RoboDK station: kr30 cnc 070119 curve 7 axis test.rdk

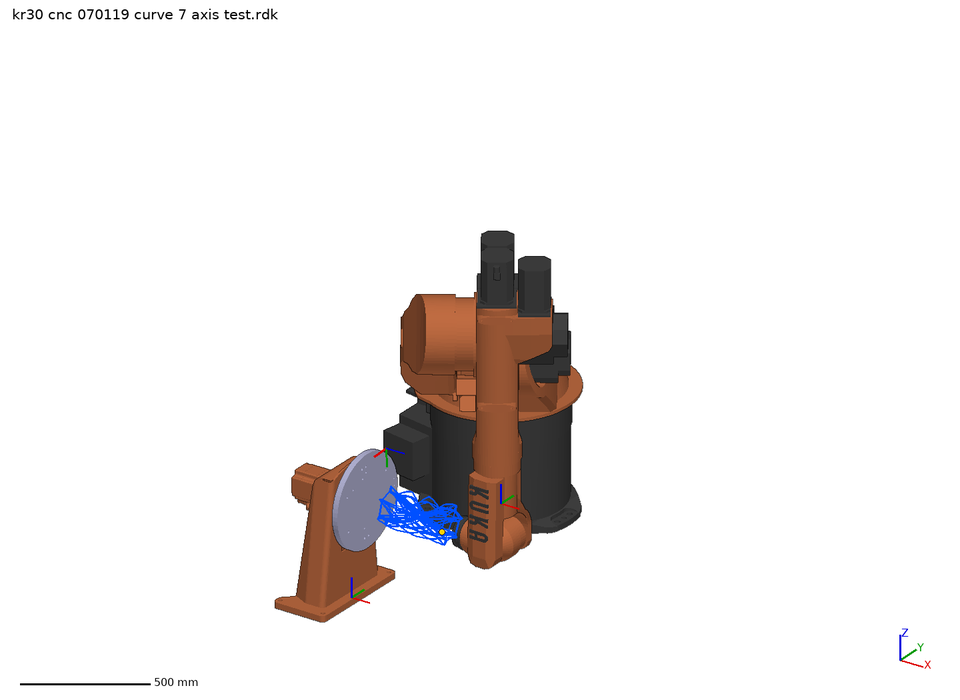
[picture v0: the station drawn from its stored meshes, robots at their saved joint values, targets as dots, program paths as lines]
Station kr30 cnc 070119 curve 7 axis test. Poses are relative to the parent item; angles as X-Y-Z fixed-axis rotations.
  - machining project Curve settings: C:/Temp/temp3/RhinoProject.stl | rotZ(0) | rotX(0)*rotY(0) | rotz(0) | onStart | onPathStart | onApproach | onPoint | onRetract | onFinish | onPathFinish
  - frame KUKA KP1 MD250 Base at (0, 1000, 0) mm
    - robot KUKA KP1 MD250: 1 axes, payload 250 kg
        modified DH rows (alpha deg, a mm, theta deg, d mm): 0, 0, 0, 0
        base shift (73.5, 0, 432) mm, rotated rx 0 ry 90 rz 0 deg
        joint limits [-3600] to [3600]; home [0]; saved at [-1886.749]
      - frame Reference Rhino at (0, -260, 100) mm
        - object RhinoPart at (0, 0, 0) mm
  - frame KUKA KR 30 HA Base at (0, 2000, 0) mm
    - robot KUKA KR 30 HA: 6 axes, payload 30 kg, reach 2033 mm, repeatability 0.05 mm, weight 665 kg
        modified DH rows (alpha deg, a mm, theta deg, d mm): 0, 0, 0, 815; -90, 350, 0, 0; 0, 850, -90, 0; -90, 145, 0, 820; 90, 0, 0, 0; -90, 0, 180, 170
        joint limits [-185, -135, -120, -350, -119, -350] to [185, 35, 158, 350, 119, 350]; home [0, -90, 90, 0, 0, 0]; saved at [55.744, -30.783, 121.676, 55.747, 89.498, 89.262]
      - tool Tool 1, TCP at (0, 0, 200) mm
  - machining project RhinoPart Settings: rotZ(0) | rotX(0)*rotY(0) | rotz(0) | onStart | onPathStart | onApproach | onPoint | onRetract | onFinish | onPathFinish
  - program RhinoPart (1340 instructions, listed below)
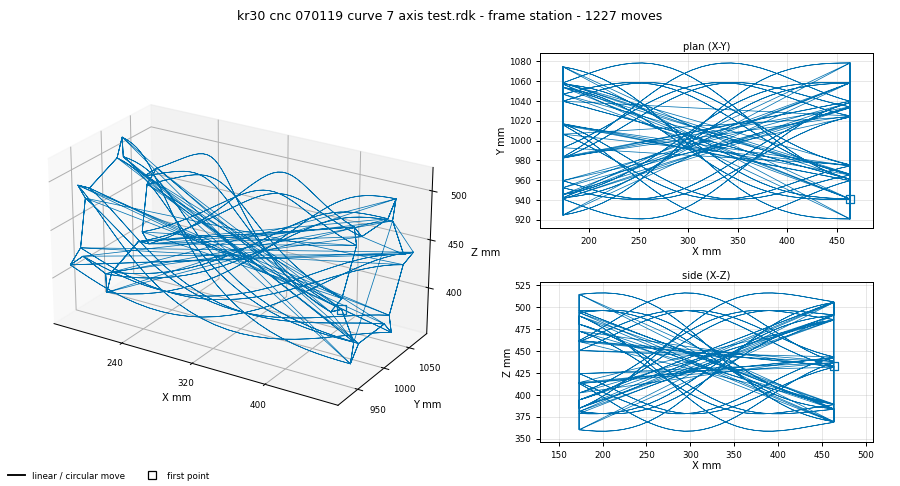
[picture p0: tool path of kr30 cnc 070119 curve 7 axis test.rdk in frame station, 1227 of 1227 moves have a stored position in this frame; points joined in program order, loops and branches not executed]

--- program RhinoPart (robot KUKA KR 30 HA) ---
  Set Ref.: Reference Rhino
  Set Tool: Tool 1
  Show Tool 1
  Set speed (1000.0 mm/s)
  MoveJ 1 to (58.93, 255.88, 290) mm, rotated rx -180 ry 0 rz -94 deg; joints [50.189, -25.769, 112.866, 50.225, 91.858, 92.231, 4.002]
  MoveL 2 to (58.93, 255.88, 290) mm, rotated rx -180 ry 0 rz -94 deg; joints [50.189, -25.769, 112.866, 50.225, 91.858, 92.231, 4.002]
  MoveL 3 to (58.93, 255.88, 290) mm, rotated rx -180 ry 0 rz -94 deg; joints [50.189, -25.769, 112.866, 50.225, 91.858, 92.231, 4.002]
  Set speed (60.0 mm/s)
  MoveL 4 to (37.11, 300.24, 290) mm, rotated rx 180 ry 0 rz -42.69 deg; joints [50.189, -26.061, 113.024, 50.228, 91.944, 92.334, -47.315]
  MoveL 5 to (-37.11, 208.63, 290) mm, rotated rx -180 ry 0 rz 144.16 deg; joints [50.189, -25.479, 112.707, 50.222, 91.774, 92.13, 125.844]
  Set speed (60.0 mm/s)
  MoveL 6 to (-58.93, 252.99, 290) mm, rotated rx -180 ry 0 rz 96.78 deg; joints [50.189, -25.75, 112.856, 50.225, 91.853, 92.224, 173.216]
  MoveL 7 to (21.11, 199.39, 290) mm, rotated rx -180 ry 0 rz -160.79 deg; joints [50.189, -25.425, 112.677, 50.221, 91.759, 92.111, 70.794]
  Set speed (60.0 mm/s)
  MoveL 8 to (34.79, 183.72, 290) mm, rotated rx -180 ry 0 rz -155.49 deg; joints [50.189, -24.101, 111.933, 50.209, 91.388, 91.665, 65.485]
  MoveL 9 to (21.11, 199.39, 290) mm, rotated rx -180 ry 0 rz -160.79 deg; joints [50.189, -25.425, 112.677, 50.221, 91.759, 92.111, 70.794]
  Set speed (60.0 mm/s)
  MoveL 10 to (-28.22, 202.67, 290) mm, rotated rx -180 ry 0 rz 153.79 deg; joints [50.189, -25.444, 112.688, 50.221, 91.764, 92.118, 116.207]
  MoveL 11 to (-43.85, 188.95, 290) mm, rotated rx -180 ry 0 rz 148.32 deg; joints [50.189, -24.124, 111.947, 50.209, 91.394, 91.673, 121.679]
  Set speed (60.0 mm/s)
  MoveL 12 to (-28.22, 202.67, 290) mm, rotated rx -180 ry 0 rz 153.79 deg; joints [50.189, -25.444, 112.688, 50.221, 91.764, 92.118, 116.207]
  MoveL 13 to (-43.85, 188.95, 290) mm, rotated rx -180 ry 0 rz 148.32 deg; joints [50.189, -24.124, 111.947, 50.209, 91.394, 91.673, 121.679]
  Set speed (60.0 mm/s)
  MoveL 14 to (-37.11, 208.63, 290) mm, rotated rx -180 ry 0 rz 144.16 deg; joints [50.189, -25.479, 112.707, 50.222, 91.774, 92.13, 125.844]
  MoveL 15 to (-78.63, 259.66, 290) mm, rotated rx -180 ry 0 rz 90.25 deg; joints [50.189, -24.451, 112.133, 50.212, 91.484, 91.781, 179.755]
  Set speed (60.0 mm/s)
  MoveL 16 to (-58.93, 252.99, 290) mm, rotated rx -180 ry 0 rz 96.78 deg; joints [50.189, -25.75, 112.856, 50.225, 91.853, 92.224, 173.216]
  MoveL 17 to (-78.63, 259.66, 290) mm, rotated rx -180 ry 0 rz 90.25 deg; joints [50.189, -24.451, 112.133, 50.212, 91.484, 91.781, 179.755]
  Set speed (60.0 mm/s)
  MoveL 18 to (-58.22, 263.67, 290) mm, rotated rx -180 ry 0 rz 86.39 deg; joints [50.189, -25.818, 112.893, 50.226, 91.873, 92.248, 183.606]
  MoveL 19 to (-30.72, 304.75, 290) mm, rotated rx -180 ry 0 rz 34.47 deg; joints [50.189, -26.092, 113.041, 50.229, 91.953, 92.345, 235.533]
  Set speed (60.0 mm/s)
  MoveL 20 to (-58.22, 263.67, 290) mm, rotated rx -180 ry 0 rz 86.39 deg; joints [50.189, -25.818, 112.893, 50.226, 91.873, 92.248, 183.606]
  MoveL 21 to (-30.72, 304.75, 290) mm, rotated rx -180 ry 0 rz 34.47 deg; joints [50.189, -26.092, 113.041, 50.229, 91.953, 92.345, 235.533]
  Set speed (60.0 mm/s)
  MoveL 22 to (-34.79, 325.15, 290) mm, rotated rx -180 ry 0 rz 28.1 deg; joints [50.189, -24.773, 112.315, 50.215, 91.574, 91.889, 241.899]
  MoveL 23 to (-21.11, 309.47, 290) mm, rotated rx 180 ry 0 rz 23.11 deg; joints [50.189, -26.125, 113.059, 50.229, 91.963, 92.356, 246.89]
  Set speed (60.0 mm/s)
  MoveL 24 to (-34.79, 325.15, 290) mm, rotated rx -180 ry 0 rz 28.1 deg; joints [50.189, -24.773, 112.315, 50.215, 91.574, 91.889, 241.899]
  MoveL 25 to (-21.11, 309.47, 290) mm, rotated rx 180 ry 0 rz 23.11 deg; joints [50.189, -26.125, 113.059, 50.229, 91.963, 92.356, 246.89]
  Set speed (60.0 mm/s)
  MoveL 26 to (28.22, 306.19, 290) mm, rotated rx -180 ry 0 rz -31.42 deg; joints [50.189, -26.102, 113.046, 50.229, 91.956, 92.348, 301.418]
  MoveL 27 to (43.85, 319.91, 290) mm, rotated rx -180 ry 0 rz -36.2 deg; joints [50.189, -24.747, 112.3, 50.214, 91.566, 91.88, 306.197]
  Set speed (60.0 mm/s)
  MoveL 28 to (28.22, 306.19, 290) mm, rotated rx -180 ry 0 rz -31.42 deg; joints [50.189, -26.102, 113.046, 50.229, 91.956, 92.348, 301.418]
  MoveL 29 to (43.85, 319.91, 290) mm, rotated rx -180 ry 0 rz -36.2 deg; joints [50.189, -24.747, 112.3, 50.214, 91.566, 91.88, 306.197]
  Set speed (60.0 mm/s)
  MoveL 30 to (37.11, 300.24, 290) mm, rotated rx 180 ry 0 rz -42.69 deg; joints [50.189, -26.061, 113.024, 50.228, 91.944, 92.334, 312.685]
  MoveL 31 to (78.63, 249.2, 290) mm, rotated rx -180 ry 0 rz -97.82 deg; joints [50.189, -24.402, 112.105, 50.211, 91.47, 91.765, 367.819]
  Set speed (60.0 mm/s)
  MoveL 32 to (58.93, 255.88, 290) mm, rotated rx 180 ry 0 rz -94 deg; joints [50.189, -25.769, 112.866, 50.225, 91.858, 92.231, 364.002]
  MoveL 33 to (78.63, 249.2, 290) mm, rotated rx -180 ry 0 rz -97.82 deg; joints [50.189, -24.402, 112.105, 50.211, 91.47, 91.765, 367.819]
  Set speed (60.0 mm/s)
  MoveL 34 to (58.22, 245.2, 290) mm, rotated rx 180 ry 0 rz -104.27 deg; joints [50.189, -25.701, 112.829, 50.224, 91.839, 92.207, 374.265]
  MoveL 35 to (30.72, 204.12, 290) mm, rotated rx 180 ry 0 rz -151.2 deg; joints [50.189, -25.453, 112.693, 50.221, 91.767, 92.121, 421.204]
  Set speed (60.0 mm/s)
  MoveL 36 to (58.22, 245.2, 290) mm, rotated rx 180 ry 0 rz -104.27 deg; joints [50.189, -25.701, 112.829, 50.224, 91.839, 92.207, 374.265]
  MoveL 37 to (30.72, 204.12, 290) mm, rotated rx 180 ry 0 rz -151.2 deg; joints [50.189, -25.453, 112.693, 50.221, 91.767, 92.121, 421.204]
  Set speed (60.0 mm/s)
  MoveL 38 to (34.79, 183.72, 290) mm, rotated rx -180 ry 0 rz -155.49 deg; joints [50.189, -24.101, 111.933, 50.209, 91.388, 91.665, 425.485]
  MoveL 39 to (-37.62, 299.82, 0) mm, rotated rx -180 ry 0 rz 43.38 deg; joints [61.476, -27.63, 125.243, 61.688, 86.373, 83.302, 586.623]
  Set speed (60.0 mm/s)
  MoveL 40 to (10.16, 312.5, 0) mm, rotated rx -180 ry 0 rz -10.95 deg; joints [61.476, -27.728, 125.294, 61.686, 86.395, 83.343, 640.953]
  MoveL 41 to (-37.62, 299.82, 0) mm, rotated rx 180 ry 0 rz 43.38 deg; joints [61.476, -27.63, 125.243, 61.688, 86.373, 83.302, 586.623]
  Set speed (60.0 mm/s)
  MoveL 42 to (-55.59, 310.29, 0) mm, rotated rx 180 ry 0 rz 47.87 deg; joints [61.476, -26.133, 124.437, 61.729, 86.045, 82.692, 582.13]
  MoveL 43 to (-45.21, 292.27, 0) mm, rotated rx -180 ry 0 rz 54.48 deg; joints [61.476, -27.574, 125.213, 61.69, 86.36, 83.279, 575.516]
  Set speed (60.0 mm/s)
  MoveL 44 to (-55.59, 310.29, 0) mm, rotated rx 180 ry 0 rz 47.87 deg; joints [61.476, -26.133, 124.437, 61.729, 86.045, 82.692, 582.13]
  MoveL 45 to (-45.21, 292.27, 0) mm, rotated rx -180 ry 0 rz 54.48 deg; joints [61.476, -27.574, 125.213, 61.69, 86.36, 83.279, 575.516]
  Set speed (60.0 mm/s)
  MoveL 46 to (-58.12, 244.54, 0) mm, rotated rx -180 ry 0 rz 104.89 deg; joints [61.476, -27.232, 125.032, 61.699, 86.284, 83.137, 525.106]
  MoveL 47 to (-76.17, 234.21, 0) mm, rotated rx 180 ry 0 rz 108.7 deg; joints [61.476, -25.73, 124.214, 61.74, 85.96, 82.533, 521.297]
  Set speed (60.0 mm/s)
  MoveL 48 to (-58.12, 244.54, 0) mm, rotated rx -180 ry 0 rz 104.89 deg; joints [61.476, -27.232, 125.032, 61.699, 86.284, 83.137, 525.106]
  MoveL 49 to (-76.17, 234.21, 0) mm, rotated rx 180 ry 0 rz 108.7 deg; joints [61.476, -25.73, 124.214, 61.74, 85.96, 82.533, 521.297]
  Set speed (60.0 mm/s)
  MoveL 50 to (-55.37, 234.2, 0) mm, rotated rx 180 ry 0 rz 114.99 deg; joints [61.476, -27.161, 124.995, 61.701, 86.268, 83.108, 515.014]
  MoveL 51 to (-20.49, 199.16, 0) mm, rotated rx -180 ry 0 rz 161.39 deg; joints [61.476, -26.93, 124.871, 61.707, 86.217, 83.013, 468.615]
  Set speed (60.0 mm/s)
  MoveL 52 to (-55.37, 234.2, 0) mm, rotated rx -180 ry 0 rz 114.99 deg; joints [61.476, -27.161, 124.995, 61.701, 86.268, 83.108, 515.014]
  MoveL 53 to (-20.49, 199.16, 0) mm, rotated rx -180 ry 0 rz 161.39 deg; joints [61.476, -26.93, 124.871, 61.707, 86.217, 83.013, 468.615]
  Set speed (60.0 mm/s)
  MoveL 54 to (-20.57, 178.36, 0) mm, rotated rx -180 ry 0 rz 165.86 deg; joints [61.476, -25.451, 124.058, 61.747, 85.902, 82.424, 464.144]
  MoveL 55 to (-10.16, 196.36, 0) mm, rotated rx -180 ry 0 rz 170.93 deg; joints [61.476, -26.912, 124.861, 61.707, 86.214, 83.006, 459.071]
  Set speed (60.0 mm/s)
  MoveL 56 to (-20.57, 178.36, 0) mm, rotated rx -180 ry 0 rz 165.86 deg; joints [61.476, -25.451, 124.058, 61.747, 85.902, 82.424, 464.144]
  MoveL 57 to (-10.16, 196.36, 0) mm, rotated rx -180 ry 0 rz 170.93 deg; joints [61.476, -26.912, 124.861, 61.707, 86.214, 83.006, 459.071]
  Set speed (60.0 mm/s)
  MoveL 58 to (37.62, 209.05, 0) mm, rotated rx 180 ry 0 rz -143.56 deg; joints [61.476, -26.994, 124.905, 61.705, 86.232, 83.039, 413.558]
  MoveL 59 to (55.59, 198.58, 0) mm, rotated rx -180 ry 0 rz -137.85 deg; joints [61.476, -25.55, 124.114, 61.745, 85.922, 82.463, 407.85]
  Set speed (60.0 mm/s)
  MoveL 60 to (37.62, 209.05, 0) mm, rotated rx -180 ry 0 rz -143.56 deg; joints [61.476, -26.994, 124.905, 61.705, 86.232, 83.039, 413.558]
  MoveL 61 to (55.59, 198.58, 0) mm, rotated rx -180 ry 0 rz -137.85 deg; joints [61.476, -25.55, 124.114, 61.745, 85.922, 82.463, 407.85]
  Set speed (60.0 mm/s)
  MoveL 62 to (45.21, 216.6, 0) mm, rotated rx -180 ry 0 rz -133.83 deg; joints [61.476, -27.044, 124.932, 61.704, 86.242, 83.059, 403.831]
  MoveL 63 to (58.12, 264.32, 0) mm, rotated rx -180 ry 0 rz -85.75 deg; joints [61.476, -27.37, 125.106, 61.695, 86.315, 83.194, 355.746]
  Set speed (60.0 mm/s)
  MoveL 64 to (45.21, 216.6, 0) mm, rotated rx -180 ry 0 rz -133.83 deg; joints [61.476, -27.044, 124.932, 61.704, 86.242, 83.059, 403.831]
  MoveL 65 to (58.12, 264.32, 0) mm, rotated rx -180 ry 0 rz -85.75 deg; joints [61.476, -27.37, 125.106, 61.695, 86.315, 83.194, 355.746]
  Set speed (60.0 mm/s)
  MoveL 66 to (76.17, 274.65, 0) mm, rotated rx -180 ry 0 rz -79.11 deg; joints [61.476, -25.94, 124.331, 61.734, 86.004, 82.616, 349.111]
  MoveL 67 to (55.37, 274.67, 0) mm, rotated rx -180 ry 0 rz -75.16 deg; joints [61.476, -27.444, 125.145, 61.693, 86.331, 83.225, 345.162]
  Set speed (60.0 mm/s)
  MoveL 68 to (76.17, 274.65, 0) mm, rotated rx -180 ry 0 rz -79.11 deg; joints [61.476, -25.94, 124.331, 61.734, 86.004, 82.616, 349.111]
  MoveL 69 to (55.37, 274.67, 0) mm, rotated rx -180 ry 0 rz -75.16 deg; joints [61.476, -27.444, 125.145, 61.693, 86.331, 83.225, 345.162]
  Set speed (60.0 mm/s)
  MoveL 70 to (20.49, 309.71, 0) mm, rotated rx -180 ry 0 rz -22.4 deg; joints [61.476, -27.706, 125.283, 61.686, 86.39, 83.334, 292.405]
  MoveL 71 to (20.57, 330.51, 0) mm, rotated rx -180 ry 0 rz -16.27 deg; joints [61.476, -26.245, 124.499, 61.726, 86.069, 82.736, 286.267]
  Set speed (60.0 mm/s)
  MoveL 72 to (20.49, 309.71, 0) mm, rotated rx -180 ry 0 rz -22.4 deg; joints [61.476, -27.706, 125.283, 61.686, 86.39, 83.334, 292.405]
  MoveL 73 to (20.57, 330.51, 0) mm, rotated rx -180 ry 0 rz -16.27 deg; joints [61.476, -26.245, 124.499, 61.726, 86.069, 82.736, 286.267]
  Set speed (60.0 mm/s)
  MoveL 74 to (10.16, 312.5, 0) mm, rotated rx 180 ry 0 rz -10.95 deg; joints [61.476, -27.728, 125.294, 61.686, 86.395, 83.343, 280.953]
  MoveL 75 to (-37.62, 299.82, 0) mm, rotated rx -180 ry 0 rz 43.38 deg; joints [61.476, -27.63, 125.243, 61.688, 86.373, 83.302, 226.623]
  Set speed (60.0 mm/s)
  MoveL 76 to (-40.85, 296.93, 10) mm, rotated rx -180 ry 0 rz 47.89 deg; joints [61.035, -27.593, 124.892, 61.233, 86.472, 83.605, 222.114]
  MoveL 77 to (-44.15, 293.5, 20) mm, rotated rx -180 ry 0 rz 52.81 deg; joints [60.599, -27.549, 124.533, 60.781, 86.578, 83.908, 217.19]
  MoveL 78 to (-47.39, 289.5, 30) mm, rotated rx -180 ry 0 rz 58.1 deg; joints [60.166, -27.499, 124.166, 60.333, 86.689, 84.21, 211.9]
  MoveL 79 to (-50.45, 284.92, 40) mm, rotated rx -180 ry 0 rz 63.71 deg; joints [59.736, -27.443, 123.791, 59.89, 86.805, 84.511, 206.29]
  MoveL 80 to (-53.21, 279.8, 50) mm, rotated rx 180 ry 0 rz 69.59 deg; joints [59.311, -27.381, 123.409, 59.45, 86.928, 84.811, 200.409]
  MoveL 81 to (-55.55, 274.16, 60) mm, rotated rx -180 ry 0 rz 75.7 deg; joints [58.889, -27.313, 123.019, 59.015, 87.055, 85.111, 194.303]
  MoveL 82 to (-57.35, 268.08, 70) mm, rotated rx -180 ry 0 rz 81.99 deg; joints [58.471, -27.241, 122.621, 58.584, 87.189, 85.41, 188.015]
  MoveL 83 to (-58.51, 261.62, 80) mm, rotated rx -180 ry 0 rz 88.41 deg; joints [58.056, -27.164, 122.217, 58.157, 87.329, 85.708, 181.589]
  MoveL 84 to (-58.95, 254.91, 90) mm, rotated rx -180 ry 0 rz 94.94 deg; joints [57.646, -27.083, 121.807, 57.734, 87.474, 86.007, 175.064]
  MoveL 85 to (-58.6, 248.05, 100) mm, rotated rx 180 ry 0 rz 101.52 deg; joints [57.239, -26.999, 121.39, 57.315, 87.626, 86.306, 168.479]
  MoveL 86 to (-57.44, 241.19, 110) mm, rotated rx 180 ry 0 rz 108.13 deg; joints [56.835, -26.914, 120.968, 56.901, 87.783, 86.605, 161.868]
  MoveL 87 to (-55.46, 234.45, 120) mm, rotated rx -180 ry 0 rz 114.74 deg; joints [56.436, -26.827, 120.541, 56.491, 87.948, 86.904, 155.264]
  MoveL 88 to (-52.68, 227.97, 130) mm, rotated rx -180 ry 0 rz 121.3 deg; joints [56.04, -26.74, 120.109, 56.086, 88.119, 87.204, 148.698]
  MoveL 89 to (-49.15, 221.88, 140) mm, rotated rx -180 ry 0 rz 127.8 deg; joints [55.647, -26.653, 119.674, 55.684, 88.296, 87.506, 142.199]
  MoveL 90 to (-44.94, 216.28, 150) mm, rotated rx -180 ry 0 rz 134.21 deg; joints [55.259, -26.567, 119.234, 55.288, 88.481, 87.808, 135.793]
  MoveL 91 to (-40.17, 211.29, 160) mm, rotated rx -180 ry 0 rz 140.49 deg; joints [54.874, -26.482, 118.791, 54.895, 88.672, 88.112, 129.508]
  MoveL 92 to (-34.94, 206.95, 170) mm, rotated rx -180 ry 0 rz 146.63 deg; joints [54.492, -26.399, 118.344, 54.508, 88.87, 88.417, 123.368]
  MoveL 93 to (-29.38, 203.32, 180) mm, rotated rx -180 ry 0 rz 152.6 deg; joints [54.114, -26.317, 117.894, 54.125, 89.076, 88.722, 117.399]
  MoveL 94 to (-23.62, 200.42, 190) mm, rotated rx -180 ry 0 rz 158.37 deg; joints [53.74, -26.237, 117.441, 53.746, 89.288, 89.029, 111.627]
  MoveL 95 to (-17.8, 198.23, 200) mm, rotated rx -180 ry 0 rz 163.92 deg; joints [53.369, -26.158, 116.984, 53.372, 89.507, 89.337, 106.077]
  MoveL 96 to (-12.04, 196.73, 210) mm, rotated rx -180 ry 0 rz 169.22 deg; joints [53.002, -26.08, 116.524, 53.003, 89.733, 89.646, 100.776]
  MoveL 97 to (-6.46, 195.84, 220) mm, rotated rx 180 ry 0 rz 174.25 deg; joints [52.638, -26.003, 116.06, 52.638, 89.966, 89.955, 95.751]
  MoveL 98 to (-1.16, 195.49, 230) mm, rotated rx 180 ry 0 rz 178.97 deg; joints [52.278, -25.926, 115.591, 52.279, 90.205, 90.264, 91.029]
  MoveL 99 to (3.78, 195.6, 240) mm, rotated rx -180 ry 0 rz -176.64 deg; joints [51.921, -25.848, 115.119, 51.924, 90.45, 90.574, 86.641]
  MoveL 100 to (8.28, 196.07, 250) mm, rotated rx 180 ry 0 rz -172.62 deg; joints [51.568, -25.768, 114.641, 51.573, 90.7, 90.883, 82.617]
  MoveL 101 to (12.3, 196.78, 260) mm, rotated rx -180 ry 0 rz -168.99 deg; joints [51.218, -25.687, 114.159, 51.228, 90.957, 91.191, 78.987]
  MoveL 102 to (15.8, 197.64, 270) mm, rotated rx -180 ry 0 rz -165.79 deg; joints [50.872, -25.603, 113.671, 50.888, 91.219, 91.499, 75.785]
  MoveL 103 to (18.74, 198.54, 280) mm, rotated rx 180 ry 0 rz -163.04 deg; joints [50.529, -25.516, 113.177, 50.552, 91.486, 91.806, 73.043]
  MoveL 104 to (21.11, 199.39, 290) mm, rotated rx -180 ry 0 rz -160.79 deg; joints [50.189, -25.425, 112.677, 50.221, 91.759, 92.111, 70.794]
  MoveL 105 to (10.16, 312.5, 0) mm, rotated rx -180 ry 0 rz -10.95 deg; joints [61.476, -27.728, 125.294, 61.686, 86.395, 83.343, -79.047]
  Set speed (60.0 mm/s)
  MoveL 106 to (-37.62, 299.82, 0) mm, rotated rx -180 ry 0 rz 43.38 deg; joints [61.476, -27.63, 125.243, 61.688, 86.373, 83.302, -133.377]
  MoveL 107 to (-28.22, 202.67, 290) mm, rotated rx 180 ry 0 rz 153.79 deg; joints [50.189, -25.444, 112.688, 50.221, 91.764, 92.118, -243.793]
  Set speed (60.0 mm/s)
  MoveL 108 to (21.11, 199.39, 290) mm, rotated rx 180 ry 0 rz -160.79 deg; joints [50.189, -25.425, 112.677, 50.221, 91.759, 92.111, -289.206]
  MoveL 109 to (-28.22, 202.67, 290) mm, rotated rx -180 ry 0 rz 153.79 deg; joints [50.189, -25.444, 112.688, 50.221, 91.764, 92.118, -243.793]
  Set speed (60.0 mm/s)
  MoveL 110 to (-30.4, 203.93, 280) mm, rotated rx 180 ry 0 rz 151.53 deg; joints [50.529, -25.548, 113.195, 50.552, 91.495, 91.817, -241.533]
  MoveL 111 to (-33, 205.58, 270) mm, rotated rx -180 ry 0 rz 148.77 deg; joints [50.872, -25.65, 113.697, 50.888, 91.232, 91.515, -238.768]
  MoveL 112 to (-35.92, 207.69, 260) mm, rotated rx 180 ry 0 rz 145.53 deg; joints [51.218, -25.752, 114.194, 51.228, 90.975, 91.214, -235.528]
  MoveL 113 to (-39.07, 210.28, 250) mm, rotated rx -180 ry 0 rz 141.84 deg; joints [51.568, -25.853, 114.688, 51.574, 90.724, 90.913, -231.841]
  MoveL 114 to (-42.34, 213.41, 240) mm, rotated rx -180 ry 0 rz 137.73 deg; joints [51.921, -25.954, 115.177, 51.924, 90.479, 90.612, -227.735]
  MoveL 115 to (-45.62, 217.1, 230) mm, rotated rx -180 ry 0 rz 133.24 deg; joints [52.278, -26.056, 115.662, 52.279, 90.241, 90.311, -223.236]
  MoveL 116 to (-48.8, 221.36, 220) mm, rotated rx -180 ry 0 rz 128.37 deg; joints [52.638, -26.158, 116.144, 52.638, 90.009, 90.011, -218.371]
  MoveL 117 to (-51.74, 226.19, 210) mm, rotated rx -180 ry 0 rz 123.16 deg; joints [53.002, -26.261, 116.622, 53.003, 89.783, 89.712, -213.164]
  MoveL 118 to (-54.33, 231.55, 200) mm, rotated rx -180 ry 0 rz 117.64 deg; joints [53.369, -26.364, 117.095, 53.371, 89.563, 89.413, -207.64]
  MoveL 119 to (-56.44, 237.4, 190) mm, rotated rx 180 ry 0 rz 111.82 deg; joints [53.74, -26.467, 117.565, 53.745, 89.351, 89.115, -201.825]
  MoveL 120 to (-57.96, 243.66, 180) mm, rotated rx -180 ry 0 rz 105.74 deg; joints [54.114, -26.571, 118.031, 54.123, 89.144, 88.817, -195.742]
  MoveL 121 to (-58.8, 250.25, 170) mm, rotated rx -180 ry 0 rz 99.42 deg; joints [54.492, -26.674, 118.493, 54.506, 88.944, 88.52, -189.418]
  MoveL 122 to (-58.89, 257.04, 160) mm, rotated rx -180 ry 0 rz 92.88 deg; joints [54.874, -26.777, 118.949, 54.893, 88.75, 88.223, -182.877]
  MoveL 123 to (-58.18, 263.92, 150) mm, rotated rx 180 ry 0 rz 86.15 deg; joints [55.259, -26.878, 119.401, 55.285, 88.562, 87.926, -176.149]
  MoveL 124 to (-56.65, 270.74, 140) mm, rotated rx -180 ry 0 rz 79.26 deg; joints [55.647, -26.976, 119.847, 55.681, 88.381, 87.629, -169.263]
  MoveL 125 to (-54.3, 277.38, 130) mm, rotated rx 180 ry 0 rz 72.25 deg; joints [56.04, -27.071, 120.286, 56.082, 88.204, 87.332, -162.251]
  MoveL 126 to (-51.17, 283.7, 120) mm, rotated rx -180 ry 0 rz 65.15 deg; joints [56.436, -27.161, 120.719, 56.487, 88.034, 87.034, -155.149]
  MoveL 127 to (-47.33, 289.58, 110) mm, rotated rx -180 ry 0 rz 57.99 deg; joints [56.835, -27.247, 121.145, 56.896, 87.868, 86.735, -147.994]
  MoveL 128 to (-42.85, 294.92, 100) mm, rotated rx -180 ry 0 rz 50.83 deg; joints [57.239, -27.326, 121.564, 57.31, 87.708, 86.434, -140.828]
  MoveL 129 to (-37.86, 299.62, 90) mm, rotated rx -180 ry 0 rz 43.7 deg; joints [57.646, -27.399, 121.974, 57.728, 87.553, 86.132, -133.695]
  MoveL 130 to (-32.46, 303.64, 80) mm, rotated rx 180 ry 0 rz 36.64 deg; joints [58.056, -27.464, 122.377, 58.151, 87.403, 85.829, -126.643]
  MoveL 131 to (-26.8, 306.94, 70) mm, rotated rx -180 ry 0 rz 29.72 deg; joints [58.471, -27.522, 122.77, 58.578, 87.258, 85.523, -119.72]
  MoveL 132 to (-21, 309.52, 60) mm, rotated rx -180 ry 0 rz 22.98 deg; joints [58.889, -27.572, 123.155, 59.009, 87.118, 85.216, -112.977]
  MoveL 133 to (-15.19, 311.39, 50) mm, rotated rx -180 ry 0 rz 16.46 deg; joints [59.311, -27.614, 123.532, 59.445, 86.984, 84.906, -106.464]
  MoveL 134 to (-9.5, 312.61, 40) mm, rotated rx -180 ry 0 rz 10.23 deg; joints [59.736, -27.649, 123.9, 59.885, 86.854, 84.595, -100.231]
  MoveL 135 to (-4.03, 313.25, 30) mm, rotated rx 180 ry 0 rz 4.33 deg; joints [60.166, -27.677, 124.26, 60.329, 86.731, 84.283, -94.327]
  MoveL 136 to (1.12, 313.37, 20) mm, rotated rx -180 ry 0 rz -1.2 deg; joints [60.599, -27.699, 124.612, 60.777, 86.612, 83.97, -88.799]
  MoveL 137 to (5.87, 313.09, 10) mm, rotated rx -180 ry 0 rz -6.31 deg; joints [61.035, -27.716, 124.957, 61.229, 86.5, 83.657, -83.692]
  MoveL 138 to (10.16, 312.5, 0) mm, rotated rx 180 ry 0 rz -10.95 deg; joints [61.476, -27.728, 125.294, 61.686, 86.395, 83.343, -79.047]
  MoveL 139 to (-37.62, 299.82, 0) mm, rotated rx -180 ry 0 rz 43.38 deg; joints [61.476, -27.63, 125.243, 61.688, 86.373, 83.302, -133.377]
  Set speed (60.0 mm/s)
  MoveL 140 to (-40.85, 296.93, 10) mm, rotated rx 180 ry 0 rz 47.89 deg; joints [61.035, -27.593, 124.892, 61.233, 86.472, 83.605, -137.886]
  MoveL 141 to (-44.15, 293.5, 20) mm, rotated rx -180 ry 0 rz 52.81 deg; joints [60.599, -27.549, 124.533, 60.781, 86.578, 83.908, -142.81]
  MoveL 142 to (-47.39, 289.5, 30) mm, rotated rx -180 ry 0 rz 58.1 deg; joints [60.166, -27.499, 124.166, 60.333, 86.689, 84.21, -148.1]
  MoveL 143 to (-50.45, 284.92, 40) mm, rotated rx -180 ry 0 rz 63.71 deg; joints [59.736, -27.443, 123.791, 59.89, 86.805, 84.511, -153.71]
  MoveL 144 to (-53.21, 279.8, 50) mm, rotated rx 180 ry 0 rz 69.59 deg; joints [59.311, -27.381, 123.409, 59.45, 86.928, 84.811, -159.591]
  MoveL 145 to (-55.55, 274.16, 60) mm, rotated rx -180 ry 0 rz 75.7 deg; joints [58.889, -27.313, 123.019, 59.015, 87.055, 85.111, -165.697]
  MoveL 146 to (-57.35, 268.08, 70) mm, rotated rx -180 ry 0 rz 81.99 deg; joints [58.471, -27.241, 122.621, 58.584, 87.189, 85.41, -171.985]
  MoveL 147 to (-58.51, 261.62, 80) mm, rotated rx -180 ry 0 rz 88.41 deg; joints [58.056, -27.164, 122.217, 58.157, 87.329, 85.708, -178.411]
  MoveL 148 to (-58.95, 254.91, 90) mm, rotated rx -180 ry 0 rz 94.94 deg; joints [57.646, -27.083, 121.807, 57.734, 87.474, 86.007, -184.936]
  MoveL 149 to (-58.6, 248.05, 100) mm, rotated rx 180 ry 0 rz 101.52 deg; joints [57.239, -26.999, 121.39, 57.315, 87.626, 86.306, -191.521]
  MoveL 150 to (-57.44, 241.19, 110) mm, rotated rx -180 ry 0 rz 108.13 deg; joints [56.835, -26.914, 120.968, 56.901, 87.783, 86.605, -198.132]
  MoveL 151 to (-55.46, 234.45, 120) mm, rotated rx -180 ry 0 rz 114.74 deg; joints [56.436, -26.827, 120.541, 56.491, 87.948, 86.904, -204.736]
  MoveL 152 to (-52.68, 227.97, 130) mm, rotated rx -180 ry 0 rz 121.3 deg; joints [56.04, -26.74, 120.109, 56.086, 88.119, 87.204, -211.302]
  MoveL 153 to (-49.15, 221.88, 140) mm, rotated rx -180 ry 0 rz 127.8 deg; joints [55.647, -26.653, 119.674, 55.684, 88.296, 87.506, -217.801]
  MoveL 154 to (-44.94, 216.28, 150) mm, rotated rx 180 ry 0 rz 134.21 deg; joints [55.259, -26.567, 119.234, 55.288, 88.481, 87.808, -224.207]
  MoveL 155 to (-40.17, 211.29, 160) mm, rotated rx -180 ry 0 rz 140.49 deg; joints [54.874, -26.482, 118.791, 54.895, 88.672, 88.112, -230.492]
  MoveL 156 to (-34.94, 206.95, 170) mm, rotated rx -180 ry 0 rz 146.63 deg; joints [54.492, -26.399, 118.344, 54.508, 88.87, 88.417, -236.632]
  MoveL 157 to (-29.38, 203.32, 180) mm, rotated rx -180 ry 0 rz 152.6 deg; joints [54.114, -26.317, 117.894, 54.125, 89.076, 88.722, -242.601]
  MoveL 158 to (-23.62, 200.42, 190) mm, rotated rx -180 ry 0 rz 158.37 deg; joints [53.74, -26.237, 117.441, 53.746, 89.288, 89.029, -248.373]
  MoveL 159 to (-17.8, 198.23, 200) mm, rotated rx -180 ry 0 rz 163.92 deg; joints [53.369, -26.158, 116.984, 53.372, 89.507, 89.337, -253.923]
  MoveL 160 to (-12.04, 196.73, 210) mm, rotated rx -180 ry 0 rz 169.22 deg; joints [53.002, -26.08, 116.524, 53.003, 89.733, 89.646, -259.224]
  MoveL 161 to (-6.46, 195.84, 220) mm, rotated rx 180 ry 0 rz 174.25 deg; joints [52.638, -26.003, 116.06, 52.638, 89.966, 89.955, -264.249]
  MoveL 162 to (-1.16, 195.49, 230) mm, rotated rx 180 ry 0 rz 178.97 deg; joints [52.278, -25.926, 115.591, 52.279, 90.205, 90.264, -268.971]
  MoveL 163 to (3.78, 195.6, 240) mm, rotated rx -180 ry 0 rz -176.64 deg; joints [51.921, -25.848, 115.119, 51.924, 90.45, 90.574, -273.359]
  MoveL 164 to (8.28, 196.07, 250) mm, rotated rx 180 ry 0 rz -172.62 deg; joints [51.568, -25.768, 114.641, 51.573, 90.7, 90.883, -277.383]
  MoveL 165 to (12.3, 196.78, 260) mm, rotated rx -180 ry 0 rz -168.99 deg; joints [51.218, -25.687, 114.159, 51.228, 90.957, 91.191, -281.013]
  MoveL 166 to (15.8, 197.64, 270) mm, rotated rx -180 ry 0 rz -165.79 deg; joints [50.872, -25.603, 113.671, 50.888, 91.219, 91.499, -284.215]
  MoveL 167 to (18.74, 198.54, 280) mm, rotated rx 180 ry 0 rz -163.04 deg; joints [50.529, -25.516, 113.177, 50.552, 91.486, 91.806, -286.957]
  MoveL 168 to (21.11, 199.39, 290) mm, rotated rx -180 ry 0 rz -160.79 deg; joints [50.189, -25.425, 112.677, 50.221, 91.759, 92.111, -289.206]
  MoveL 169 to (34.79, 183.72, 290) mm, rotated rx -180 ry 0 rz -155.49 deg; joints [50.189, -24.101, 111.933, 50.209, 91.388, 91.665, -294.515]
  Set speed (60.0 mm/s)
  MoveL 170 to (21.11, 199.39, 290) mm, rotated rx -180 ry 0 rz -160.79 deg; joints [50.189, -25.425, 112.677, 50.221, 91.759, 92.111, -289.206]
  MoveL 171 to (-55.59, 310.29, 0) mm, rotated rx 180 ry 0 rz 47.87 deg; joints [61.476, -26.133, 124.437, 61.729, 86.045, 82.692, -137.87]
  Set speed (60.0 mm/s)
  MoveL 172 to (-37.62, 299.82, 0) mm, rotated rx -180 ry 0 rz 43.38 deg; joints [61.476, -27.63, 125.243, 61.688, 86.373, 83.302, -133.377]
  MoveL 173 to (34.79, 183.72, 290) mm, rotated rx -180 ry 0 rz -155.49 deg; joints [50.189, -24.101, 111.933, 50.209, 91.388, 91.665, -294.515]
  Set speed (60.0 mm/s)
  MoveL 174 to (31.73, 182.3, 280) mm, rotated rx -180 ry 0 rz -157.79 deg; joints [50.529, -24.186, 112.431, 50.542, 91.116, 91.355, -292.214]
  MoveL 175 to (27.92, 180.74, 270) mm, rotated rx -180 ry 0 rz -160.59 deg; joints [50.872, -24.267, 112.922, 50.879, 90.849, 91.043, -289.407]
  MoveL 176 to (23.38, 179.17, 260) mm, rotated rx 180 ry 0 rz -163.87 deg; joints [51.218, -24.344, 113.407, 51.222, 90.587, 90.73, -286.13]
  MoveL 177 to (18.11, 177.74, 250) mm, rotated rx 180 ry 0 rz -167.58 deg; joints [51.568, -24.418, 113.886, 51.569, 90.331, 90.417, -282.417]
  MoveL 178 to (12.17, 176.57, 240) mm, rotated rx -180 ry 0 rz -171.7 deg; joints [51.921, -24.49, 114.361, 51.921, 90.08, 90.102, -278.3]
  MoveL 179 to (5.61, 175.83, 230) mm, rotated rx -180 ry 0 rz -176.19 deg; joints [52.278, -24.561, 114.83, 52.278, 89.835, 89.787, -273.813]
  MoveL 180 to (-1.49, 175.64, 220) mm, rotated rx -180 ry 0 rz 178.99 deg; joints [52.638, -24.631, 115.295, 52.64, 89.597, 89.472, -268.987]
  MoveL 181 to (-9.03, 176.15, 210) mm, rotated rx -180 ry 0 rz 173.85 deg; joints [53.002, -24.7, 115.756, 53.007, 89.365, 89.157, -263.854]
  MoveL 182 to (-16.88, 177.46, 200) mm, rotated rx -180 ry 0 rz 168.44 deg; joints [53.369, -24.771, 116.213, 53.378, 89.14, 88.843, -258.444]
  MoveL 183 to (-24.89, 179.66, 190) mm, rotated rx 180 ry 0 rz 162.78 deg; joints [53.74, -24.842, 116.666, 53.754, 88.921, 88.529, -252.785]
  MoveL 184 to (-32.91, 182.83, 180) mm, rotated rx -180 ry 0 rz 156.91 deg; joints [54.114, -24.914, 117.116, 54.134, 88.709, 88.215, -246.906]
  MoveL 185 to (-40.75, 186.98, 170) mm, rotated rx -180 ry 0 rz 150.84 deg; joints [54.492, -24.988, 117.563, 54.52, 88.505, 87.903, -240.836]
  MoveL 186 to (-48.24, 192.12, 160) mm, rotated rx 180 ry 0 rz 144.6 deg; joints [54.874, -25.064, 118.007, 54.909, 88.307, 87.592, -234.602]
  MoveL 187 to (-55.2, 198.19, 150) mm, rotated rx -180 ry 0 rz 138.23 deg; joints [55.259, -25.142, 118.448, 55.303, 88.117, 87.282, -228.231]
  MoveL 188 to (-61.48, 205.13, 140) mm, rotated rx 180 ry 0 rz 131.75 deg; joints [55.647, -25.221, 118.885, 55.702, 87.933, 86.973, -221.752]
  MoveL 189 to (-66.92, 212.81, 130) mm, rotated rx -180 ry 0 rz 125.19 deg; joints [56.04, -25.301, 119.318, 56.105, 87.757, 86.666, -215.192]
  MoveL 190 to (-71.41, 221.1, 120) mm, rotated rx 180 ry 0 rz 118.58 deg; joints [56.436, -25.381, 119.748, 56.512, 87.587, 86.359, -208.581]
  MoveL 191 to (-74.87, 229.83, 110) mm, rotated rx -180 ry 0 rz 111.95 deg; joints [56.835, -25.462, 120.173, 56.924, 87.425, 86.053, -201.949]
  MoveL 192 to (-77.24, 238.83, 100) mm, rotated rx -180 ry 0 rz 105.33 deg; joints [57.239, -25.541, 120.594, 57.34, 87.269, 85.748, -195.327]
  MoveL 193 to (-78.53, 247.91, 90) mm, rotated rx -180 ry 0 rz 98.75 deg; joints [57.646, -25.62, 121.009, 57.76, 87.119, 85.443, -188.75]
  MoveL 194 to (-78.77, 256.9, 80) mm, rotated rx -180 ry 0 rz 92.25 deg; joints [58.056, -25.695, 121.418, 58.185, 86.976, 85.139, -182.251]
  MoveL 195 to (-78, 265.63, 70) mm, rotated rx -180 ry 0 rz 85.87 deg; joints [58.471, -25.767, 121.821, 58.614, 86.839, 84.835, -175.868]
  MoveL 196 to (-76.35, 273.96, 60) mm, rotated rx -180 ry 0 rz 79.64 deg; joints [58.889, -25.836, 122.218, 59.046, 86.707, 84.53, -169.641]
  MoveL 197 to (-73.92, 281.75, 50) mm, rotated rx 180 ry 0 rz 73.61 deg; joints [59.311, -25.899, 122.607, 59.483, 86.582, 84.225, -163.608]
  MoveL 198 to (-70.87, 288.9, 40) mm, rotated rx -180 ry 0 rz 67.81 deg; joints [59.736, -25.957, 122.988, 59.924, 86.463, 83.919, -157.812]
  MoveL 199 to (-67.34, 295.36, 30) mm, rotated rx -180 ry 0 rz 62.3 deg; joints [60.166, -26.01, 123.363, 60.369, 86.35, 83.613, -152.296]
  MoveL 200 to (-63.51, 301.08, 20) mm, rotated rx -180 ry 0 rz 57.1 deg; joints [60.599, -26.057, 123.729, 60.819, 86.242, 83.307, -147.105]
  MoveL 201 to (-59.54, 306.05, 10) mm, rotated rx -180 ry 0 rz 52.28 deg; joints [61.035, -26.098, 124.087, 61.272, 86.141, 82.999, -142.281]
  MoveL 202 to (-55.59, 310.29, 0) mm, rotated rx -180 ry 0 rz 47.87 deg; joints [61.476, -26.133, 124.437, 61.729, 86.045, 82.692, -137.87]
  MoveL 203 to (34.79, 183.72, 290) mm, rotated rx -180 ry 0 rz -155.49 deg; joints [50.189, -24.101, 111.933, 50.209, 91.388, 91.665, -294.515]
  Set speed (60.0 mm/s)
  MoveL 204 to (30.72, 204.12, 290) mm, rotated rx -180 ry 0 rz -151.2 deg; joints [50.189, -25.453, 112.693, 50.221, 91.767, 92.121, -298.796]
  MoveL 205 to (-55.59, 310.29, 0) mm, rotated rx 180 ry 0 rz 47.87 deg; joints [61.476, -26.133, 124.437, 61.729, 86.045, 82.692, -137.87]
  Set speed (60.0 mm/s)
  MoveL 206 to (-45.21, 292.27, 0) mm, rotated rx -180 ry 0 rz 54.48 deg; joints [61.476, -27.574, 125.213, 61.69, 86.36, 83.279, -144.484]
  MoveL 207 to (-55.59, 310.29, 0) mm, rotated rx -180 ry 0 rz 47.87 deg; joints [61.476, -26.133, 124.437, 61.729, 86.045, 82.692, -137.87]
  Set speed (60.0 mm/s)
  MoveL 208 to (-59.54, 306.05, 10) mm, rotated rx -180 ry 0 rz 52.28 deg; joints [61.035, -26.098, 124.087, 61.272, 86.141, 82.999, -142.281]
  MoveL 209 to (-63.51, 301.08, 20) mm, rotated rx 180 ry 0 rz 57.1 deg; joints [60.599, -26.057, 123.729, 60.819, 86.242, 83.307, -147.105]
  MoveL 210 to (-67.34, 295.36, 30) mm, rotated rx -180 ry 0 rz 62.3 deg; joints [60.166, -26.01, 123.363, 60.369, 86.35, 83.613, -152.296]
  MoveL 211 to (-70.87, 288.9, 40) mm, rotated rx -180 ry 0 rz 67.81 deg; joints [59.736, -25.957, 122.988, 59.924, 86.463, 83.919, -157.812]
  MoveL 212 to (-73.92, 281.75, 50) mm, rotated rx -180 ry 0 rz 73.61 deg; joints [59.311, -25.899, 122.607, 59.483, 86.582, 84.225, -163.608]
  MoveL 213 to (-76.35, 273.96, 60) mm, rotated rx 180 ry 0 rz 79.64 deg; joints [58.889, -25.836, 122.218, 59.046, 86.707, 84.53, -169.641]
  MoveL 214 to (-78, 265.63, 70) mm, rotated rx -180 ry 0 rz 85.87 deg; joints [58.471, -25.767, 121.821, 58.614, 86.839, 84.835, -175.868]
  MoveL 215 to (-78.77, 256.9, 80) mm, rotated rx -180 ry 0 rz 92.25 deg; joints [58.056, -25.695, 121.418, 58.185, 86.976, 85.139, -182.251]
  MoveL 216 to (-78.53, 247.91, 90) mm, rotated rx -180 ry 0 rz 98.75 deg; joints [57.646, -25.62, 121.009, 57.76, 87.119, 85.443, -188.75]
  MoveL 217 to (-77.24, 238.83, 100) mm, rotated rx -180 ry 0 rz 105.33 deg; joints [57.239, -25.541, 120.594, 57.34, 87.269, 85.748, -195.327]
  MoveL 218 to (-74.87, 229.83, 110) mm, rotated rx -180 ry 0 rz 111.95 deg; joints [56.835, -25.462, 120.173, 56.924, 87.425, 86.053, -201.949]
  MoveL 219 to (-71.41, 221.1, 120) mm, rotated rx -180 ry 0 rz 118.58 deg; joints [56.436, -25.381, 119.748, 56.512, 87.587, 86.359, -208.581]
  MoveL 220 to (-66.92, 212.81, 130) mm, rotated rx -180 ry 0 rz 125.19 deg; joints [56.04, -25.301, 119.318, 56.105, 87.757, 86.666, -215.192]
  MoveL 221 to (-61.48, 205.13, 140) mm, rotated rx 180 ry 0 rz 131.75 deg; joints [55.647, -25.221, 118.885, 55.702, 87.933, 86.973, -221.752]
  MoveL 222 to (-55.2, 198.19, 150) mm, rotated rx -180 ry 0 rz 138.23 deg; joints [55.259, -25.142, 118.448, 55.303, 88.117, 87.282, -228.231]
  MoveL 223 to (-48.24, 192.12, 160) mm, rotated rx -180 ry 0 rz 144.6 deg; joints [54.874, -25.064, 118.007, 54.909, 88.307, 87.592, -234.602]
  MoveL 224 to (-40.75, 186.98, 170) mm, rotated rx 180 ry 0 rz 150.84 deg; joints [54.492, -24.988, 117.563, 54.52, 88.505, 87.903, -240.836]
  MoveL 225 to (-32.91, 182.83, 180) mm, rotated rx -180 ry 0 rz 156.91 deg; joints [54.114, -24.914, 117.116, 54.134, 88.709, 88.215, -246.906]
  MoveL 226 to (-24.89, 179.66, 190) mm, rotated rx 180 ry 0 rz 162.78 deg; joints [53.74, -24.842, 116.666, 53.754, 88.921, 88.529, -252.785]
  MoveL 227 to (-16.88, 177.46, 200) mm, rotated rx -180 ry 0 rz 168.44 deg; joints [53.369, -24.771, 116.213, 53.378, 89.14, 88.843, -258.444]
  MoveL 228 to (-9.03, 176.15, 210) mm, rotated rx -180 ry 0 rz 173.85 deg; joints [53.002, -24.7, 115.756, 53.007, 89.365, 89.157, -263.854]
  MoveL 229 to (-1.49, 175.64, 220) mm, rotated rx -180 ry 0 rz 178.99 deg; joints [52.638, -24.631, 115.295, 52.64, 89.597, 89.472, -268.987]
  MoveL 230 to (5.61, 175.83, 230) mm, rotated rx -180 ry 0 rz -176.19 deg; joints [52.278, -24.561, 114.83, 52.278, 89.835, 89.787, -273.813]
  MoveL 231 to (12.17, 176.57, 240) mm, rotated rx -180 ry 0 rz -171.7 deg; joints [51.921, -24.49, 114.361, 51.921, 90.08, 90.102, -278.3]
  MoveL 232 to (18.11, 177.74, 250) mm, rotated rx -180 ry 0 rz -167.58 deg; joints [51.568, -24.418, 113.886, 51.569, 90.331, 90.417, -282.417]
  MoveL 233 to (23.38, 179.17, 260) mm, rotated rx 180 ry 0 rz -163.87 deg; joints [51.218, -24.344, 113.407, 51.222, 90.587, 90.73, -286.13]
  MoveL 234 to (27.92, 180.74, 270) mm, rotated rx -180 ry 0 rz -160.59 deg; joints [50.872, -24.267, 112.922, 50.879, 90.849, 91.043, -289.407]
  MoveL 235 to (31.73, 182.3, 280) mm, rotated rx 180 ry 0 rz -157.79 deg; joints [50.529, -24.186, 112.431, 50.542, 91.116, 91.355, -292.214]
  MoveL 236 to (34.79, 183.72, 290) mm, rotated rx -180 ry 0 rz -155.49 deg; joints [50.189, -24.101, 111.933, 50.209, 91.388, 91.665, -294.515]
  MoveL 237 to (30.72, 204.12, 290) mm, rotated rx -180 ry 0 rz -151.2 deg; joints [50.189, -25.453, 112.693, 50.221, 91.767, 92.121, -298.796]
  Set speed (60.0 mm/s)
  MoveL 238 to (28.54, 202.85, 280) mm, rotated rx 180 ry 0 rz -153.47 deg; joints [50.529, -25.541, 113.191, 50.552, 91.494, 91.814, -296.535]
  MoveL 239 to (25.81, 201.43, 270) mm, rotated rx -180 ry 0 rz -156.22 deg; joints [50.872, -25.625, 113.683, 50.888, 91.225, 91.507, -293.779]
  MoveL 240 to (22.53, 199.96, 260) mm, rotated rx 180 ry 0 rz -159.44 deg; joints [51.218, -25.706, 114.169, 51.228, 90.962, 91.198, -290.563]
  MoveL 241 to (18.7, 198.53, 250) mm, rotated rx -180 ry 0 rz -163.08 deg; joints [51.568, -25.783, 114.649, 51.573, 90.705, 90.888, -286.921]
  MoveL 242 to (14.35, 197.26, 240) mm, rotated rx 180 ry 0 rz -167.11 deg; joints [51.921, -25.857, 115.124, 51.924, 90.452, 90.577, -282.886]
  MoveL 243 to (9.52, 196.26, 230) mm, rotated rx 180 ry 0 rz -171.51 deg; joints [52.278, -25.93, 115.594, 52.279, 90.206, 90.266, -278.492]
  MoveL 244 to (4.24, 195.64, 220) mm, rotated rx 180 ry 0 rz -176.23 deg; joints [52.638, -26.002, 116.059, 52.638, 89.965, 89.955, -273.769]
  MoveL 245 to (-1.41, 195.5, 210) mm, rotated rx -180 ry 0 rz 178.75 deg; joints [53.002, -26.073, 116.52, 53.003, 89.731, 89.643, -268.748]
  MoveL 246 to (-7.35, 195.94, 200) mm, rotated rx -180 ry 0 rz 173.46 deg; joints [53.369, -26.144, 116.976, 53.372, 89.504, 89.332, -263.458]
  MoveL 247 to (-13.47, 197.04, 190) mm, rotated rx -180 ry 0 rz 167.93 deg; joints [53.74, -26.217, 117.43, 53.746, 89.283, 89.022, -257.927]
  MoveL 248 to (-19.65, 198.85, 180) mm, rotated rx -180 ry 0 rz 162.18 deg; joints [54.114, -26.29, 117.879, 54.125, 89.069, 88.712, -252.183]
  MoveL 249 to (-25.78, 201.42, 170) mm, rotated rx -180 ry 0 rz 156.25 deg; joints [54.492, -26.365, 118.326, 54.508, 88.861, 88.404, -246.252]
  MoveL 250 to (-31.7, 204.73, 160) mm, rotated rx -180 ry 0 rz 150.16 deg; joints [54.874, -26.442, 118.769, 54.896, 88.661, 88.097, -240.159]
  MoveL 251 to (-37.3, 208.79, 150) mm, rotated rx 180 ry 0 rz 143.93 deg; joints [55.259, -26.52, 119.209, 55.288, 88.468, 87.79, -233.93]
  MoveL 252 to (-42.45, 213.53, 140) mm, rotated rx 180 ry 0 rz 137.59 deg; joints [55.647, -26.601, 119.645, 55.685, 88.282, 87.486, -227.591]
  MoveL 253 to (-47.02, 218.88, 130) mm, rotated rx -180 ry 0 rz 131.17 deg; joints [56.04, -26.682, 120.078, 56.086, 88.104, 87.182, -221.168]
  MoveL 254 to (-50.93, 224.75, 120) mm, rotated rx 180 ry 0 rz 124.69 deg; joints [56.436, -26.764, 120.507, 56.492, 87.932, 86.88, -214.687]
  MoveL 255 to (-54.1, 231.02, 110) mm, rotated rx -180 ry 0 rz 118.18 deg; joints [56.835, -26.847, 120.932, 56.902, 87.767, 86.579, -208.176]
  MoveL 256 to (-56.49, 237.56, 100) mm, rotated rx -180 ry 0 rz 111.66 deg; joints [57.239, -26.93, 121.353, 57.316, 87.608, 86.278, -201.664]
  MoveL 257 to (-58.06, 244.24, 90) mm, rotated rx -180 ry 0 rz 105.18 deg; joints [57.646, -27.011, 121.768, 57.735, 87.456, 85.979, -195.184]
  MoveL 258 to (-58.85, 250.92, 80) mm, rotated rx -180 ry 0 rz 98.77 deg; joints [58.056, -27.09, 122.178, 58.158, 87.311, 85.679, -188.767]
  MoveL 259 to (-58.87, 257.48, 70) mm, rotated rx -180 ry 0 rz 92.45 deg; joints [58.471, -27.167, 122.582, 58.585, 87.171, 85.38, -182.451]
  MoveL 260 to (-58.2, 263.79, 60) mm, rotated rx -180 ry 0 rz 86.27 deg; joints [58.889, -27.24, 122.98, 59.016, 87.038, 85.081, -176.272]
  MoveL 261 to (-56.92, 269.76, 50) mm, rotated rx 180 ry 0 rz 80.27 deg; joints [59.311, -27.309, 123.371, 59.452, 86.91, 84.782, -170.271]
  MoveL 262 to (-55.13, 275.3, 40) mm, rotated rx 180 ry 0 rz 74.49 deg; joints [59.736, -27.373, 123.755, 59.891, 86.789, 84.483, -164.491]
  MoveL 263 to (-52.95, 280.35, 30) mm, rotated rx -180 ry 0 rz 68.98 deg; joints [60.166, -27.432, 124.131, 60.335, 86.673, 84.182, -158.976]
  MoveL 264 to (-50.48, 284.87, 20) mm, rotated rx -180 ry 0 rz 63.77 deg; joints [60.599, -27.485, 124.5, 60.782, 86.563, 83.882, -153.772]
  MoveL 265 to (-47.86, 288.84, 10) mm, rotated rx -180 ry 0 rz 58.93 deg; joints [61.035, -27.532, 124.86, 61.234, 86.459, 83.58, -148.926]
  MoveL 266 to (-45.21, 292.27, 0) mm, rotated rx -180 ry 0 rz 54.48 deg; joints [61.476, -27.574, 125.213, 61.69, 86.36, 83.279, -144.484]
  MoveL 267 to (30.72, 204.12, 290) mm, rotated rx -180 ry 0 rz -151.2 deg; joints [50.189, -25.453, 112.693, 50.221, 91.767, 92.121, -298.796]
  Set speed (60.0 mm/s)
  MoveL 268 to (58.22, 245.2, 290) mm, rotated rx -180 ry 0 rz -104.27 deg; joints [50.189, -25.701, 112.829, 50.224, 91.839, 92.207, -345.735]
  MoveL 269 to (-45.21, 292.27, 0) mm, rotated rx -180 ry 0 rz 54.48 deg; joints [61.476, -27.574, 125.213, 61.69, 86.36, 83.279, -504.484]
  Set speed (60.0 mm/s)
  MoveL 270 to (-58.12, 244.54, 0) mm, rotated rx 180 ry 0 rz 104.89 deg; joints [61.476, -27.232, 125.032, 61.699, 86.284, 83.137, -554.894]
  MoveL 271 to (-45.21, 292.27, 0) mm, rotated rx -180 ry 0 rz 54.48 deg; joints [61.476, -27.574, 125.213, 61.69, 86.36, 83.279, -504.484]
  Set speed (60.0 mm/s)
  MoveL 272 to (-47.86, 288.84, 10) mm, rotated rx -180 ry 0 rz 58.93 deg; joints [61.035, -27.532, 124.86, 61.234, 86.459, 83.58, -508.926]
  MoveL 273 to (-50.48, 284.87, 20) mm, rotated rx -180 ry 0 rz 63.77 deg; joints [60.599, -27.485, 124.5, 60.782, 86.563, 83.882, -513.772]
  MoveL 274 to (-52.95, 280.35, 30) mm, rotated rx 180 ry 0 rz 68.98 deg; joints [60.166, -27.432, 124.131, 60.335, 86.673, 84.182, -518.976]
  MoveL 275 to (-55.13, 275.3, 40) mm, rotated rx -180 ry 0 rz 74.49 deg; joints [59.736, -27.373, 123.755, 59.891, 86.789, 84.483, -524.491]
  MoveL 276 to (-56.92, 269.76, 50) mm, rotated rx -180 ry 0 rz 80.27 deg; joints [59.311, -27.309, 123.371, 59.452, 86.91, 84.782, -530.271]
  MoveL 277 to (-58.2, 263.79, 60) mm, rotated rx -180 ry 0 rz 86.27 deg; joints [58.889, -27.24, 122.98, 59.016, 87.038, 85.081, -536.272]
  MoveL 278 to (-58.87, 257.48, 70) mm, rotated rx -180 ry 0 rz 92.45 deg; joints [58.471, -27.167, 122.582, 58.585, 87.171, 85.38, -542.451]
  MoveL 279 to (-58.85, 250.92, 80) mm, rotated rx 180 ry 0 rz 98.77 deg; joints [58.056, -27.09, 122.178, 58.158, 87.311, 85.679, -548.767]
  MoveL 280 to (-58.06, 244.24, 90) mm, rotated rx -180 ry 0 rz 105.18 deg; joints [57.646, -27.011, 121.768, 57.735, 87.456, 85.979, -555.184]
  MoveL 281 to (-56.49, 237.56, 100) mm, rotated rx -180 ry 0 rz 111.66 deg; joints [57.239, -26.93, 121.353, 57.316, 87.608, 86.278, -561.664]
  MoveL 282 to (-54.1, 231.02, 110) mm, rotated rx -180 ry 0 rz 118.18 deg; joints [56.835, -26.847, 120.932, 56.902, 87.767, 86.579, -568.176]
  MoveL 283 to (-50.93, 224.75, 120) mm, rotated rx -180 ry 0 rz 124.69 deg; joints [56.436, -26.764, 120.507, 56.492, 87.932, 86.88, -574.687]
  MoveL 284 to (-47.02, 218.88, 130) mm, rotated rx -180 ry 0 rz 131.17 deg; joints [56.04, -26.682, 120.078, 56.086, 88.104, 87.182, -581.168]
  MoveL 285 to (-42.45, 213.53, 140) mm, rotated rx -180 ry 0 rz 137.59 deg; joints [55.647, -26.601, 119.645, 55.685, 88.282, 87.486, -587.591]
  MoveL 286 to (-37.3, 208.79, 150) mm, rotated rx -180 ry 0 rz 143.93 deg; joints [55.259, -26.52, 119.209, 55.288, 88.468, 87.79, -593.93]
  MoveL 287 to (-31.7, 204.73, 160) mm, rotated rx -180 ry 0 rz 150.16 deg; joints [54.874, -26.442, 118.769, 54.896, 88.661, 88.097, -600.159]
  MoveL 288 to (-25.78, 201.42, 170) mm, rotated rx -180 ry 0 rz 156.25 deg; joints [54.492, -26.365, 118.326, 54.508, 88.861, 88.404, -606.252]
  MoveL 289 to (-19.65, 198.85, 180) mm, rotated rx -180 ry 0 rz 162.18 deg; joints [54.114, -26.29, 117.879, 54.125, 89.069, 88.712, -612.183]
  MoveL 290 to (-13.47, 197.04, 190) mm, rotated rx -180 ry 0 rz 167.93 deg; joints [53.74, -26.217, 117.43, 53.746, 89.283, 89.022, -617.927]
  MoveL 291 to (-7.35, 195.94, 200) mm, rotated rx -180 ry 0 rz 173.46 deg; joints [53.369, -26.144, 116.976, 53.372, 89.504, 89.332, -623.458]
  MoveL 292 to (-1.41, 195.5, 210) mm, rotated rx 180 ry 0 rz 178.75 deg; joints [53.002, -26.073, 116.52, 53.003, 89.731, 89.643, -628.748]
  MoveL 293 to (4.24, 195.64, 220) mm, rotated rx 180 ry 0 rz -176.23 deg; joints [52.638, -26.002, 116.059, 52.638, 89.965, 89.955, -633.769]
  MoveL 294 to (9.52, 196.26, 230) mm, rotated rx -180 ry 0 rz -171.51 deg; joints [52.278, -25.93, 115.594, 52.279, 90.206, 90.266, -638.492]
  MoveL 295 to (14.35, 197.26, 240) mm, rotated rx -180 ry 0 rz -167.11 deg; joints [51.921, -25.857, 115.124, 51.924, 90.452, 90.577, -642.886]
  MoveL 296 to (18.7, 198.53, 250) mm, rotated rx -180 ry 0 rz -163.08 deg; joints [51.568, -25.783, 114.649, 51.573, 90.705, 90.888, -646.921]
  MoveL 297 to (22.53, 199.96, 260) mm, rotated rx -180 ry 0 rz -159.44 deg; joints [51.218, -25.706, 114.169, 51.228, 90.962, 91.198, -650.563]
  MoveL 298 to (25.81, 201.43, 270) mm, rotated rx -180 ry 0 rz -156.22 deg; joints [50.872, -25.625, 113.683, 50.888, 91.225, 91.507, -653.779]
  MoveL 299 to (28.54, 202.85, 280) mm, rotated rx 180 ry 0 rz -153.47 deg; joints [50.529, -25.541, 113.191, 50.552, 91.494, 91.814, -656.535]
  MoveL 300 to (30.72, 204.12, 290) mm, rotated rx -180 ry 0 rz -151.2 deg; joints [50.189, -25.453, 112.693, 50.221, 91.767, 92.121, -658.796]
  MoveL 301 to (58.22, 245.2, 290) mm, rotated rx 180 ry 0 rz -104.27 deg; joints [50.189, -25.701, 112.829, 50.224, 91.839, 92.207, -705.735]
  Set speed (60.0 mm/s)
  MoveL 302 to (57.77, 242.72, 280) mm, rotated rx -180 ry 0 rz -106.66 deg; joints [50.529, -25.783, 113.323, 50.554, 91.563, 91.899, -703.345]
  MoveL 303 to (57.08, 239.72, 270) mm, rotated rx -180 ry 0 rz -109.56 deg; joints [50.872, -25.858, 113.81, 50.89, 91.292, 91.588, -700.439]
  MoveL 304 to (56.08, 236.26, 260) mm, rotated rx 180 ry 0 rz -112.94 deg; joints [51.218, -25.926, 114.289, 51.23, 91.025, 91.276, -697.057]
  MoveL 305 to (54.69, 232.42, 250) mm, rotated rx -180 ry 0 rz -116.76 deg; joints [51.568, -25.988, 114.762, 51.574, 90.763, 90.961, -693.242]
  MoveL 306 to (52.84, 228.29, 240) mm, rotated rx 180 ry 0 rz -120.97 deg; joints [51.921, -26.046, 115.227, 51.924, 90.505, 90.645, -689.031]
  MoveL 307 to (50.46, 223.96, 230) mm, rotated rx -180 ry 0 rz -125.53 deg; joints [52.278, -26.098, 115.685, 52.279, 90.253, 90.326, -684.466]
  MoveL 308 to (47.51, 219.54, 220) mm, rotated rx 180 ry 0 rz -130.42 deg; joints [52.638, -26.147, 116.138, 52.638, 90.005, 90.007, -679.584]
  MoveL 309 to (43.95, 215.15, 210) mm, rotated rx -180 ry 0 rz -135.58 deg; joints [53.002, -26.192, 116.584, 53.003, 89.764, 89.687, -674.422]
  MoveL 310 to (39.77, 210.92, 200) mm, rotated rx 180 ry 0 rz -140.98 deg; joints [53.369, -26.235, 117.026, 53.372, 89.528, 89.366, -669.016]
  MoveL 311 to (34.96, 206.97, 190) mm, rotated rx 180 ry 0 rz -146.6 deg; joints [53.74, -26.277, 117.462, 53.746, 89.299, 89.044, -663.399]
  MoveL 312 to (29.57, 203.44, 180) mm, rotated rx 180 ry 0 rz -152.4 deg; joints [54.114, -26.318, 117.894, 54.125, 89.076, 88.723, -657.602]
  MoveL 313 to (23.65, 200.44, 170) mm, rotated rx -180 ry 0 rz -158.34 deg; joints [54.492, -26.359, 118.322, 54.508, 88.86, 88.402, -651.658]
  MoveL 314 to (17.28, 198.07, 160) mm, rotated rx -180 ry 0 rz -164.41 deg; joints [54.874, -26.401, 118.747, 54.896, 88.651, 88.081, -645.594]
  MoveL 315 to (10.57, 196.44, 150) mm, rotated rx -180 ry 0 rz -170.56 deg; joints [55.259, -26.444, 119.167, 55.289, 88.449, 87.762, -639.438]
  MoveL 316 to (3.62, 195.59, 140) mm, rotated rx 180 ry 0 rz -176.78 deg; joints [55.647, -26.489, 119.585, 55.686, 88.254, 87.443, -633.219]
  MoveL 317 to (-3.42, 195.58, 130) mm, rotated rx -180 ry 0 rz 176.96 deg; joints [56.04, -26.536, 120, 56.088, 88.066, 87.126, -626.961]
  MoveL 318 to (-10.42, 196.41, 120) mm, rotated rx -180 ry 0 rz 170.69 deg; joints [56.436, -26.586, 120.411, 56.495, 87.886, 86.811, -620.691]
  MoveL 319 to (-17.25, 198.06, 110) mm, rotated rx 180 ry 0 rz 164.44 deg; joints [56.835, -26.638, 120.82, 56.905, 87.714, 86.497, -614.435]
  MoveL 320 to (-23.78, 200.49, 100) mm, rotated rx -180 ry 0 rz 158.22 deg; joints [57.239, -26.692, 121.225, 57.32, 87.549, 86.185, -608.22]
  MoveL 321 to (-29.89, 203.62, 90) mm, rotated rx -180 ry 0 rz 152.07 deg; joints [57.646, -26.747, 121.627, 57.74, 87.391, 85.875, -602.072]
  MoveL 322 to (-35.48, 207.36, 80) mm, rotated rx -180 ry 0 rz 146.02 deg; joints [58.056, -26.805, 122.025, 58.163, 87.241, 85.567, -596.02]
  MoveL 323 to (-40.49, 211.59, 70) mm, rotated rx -180 ry 0 rz 140.09 deg; joints [58.471, -26.863, 122.42, 58.591, 87.097, 85.259, -590.093]
  MoveL 324 to (-44.86, 216.19, 60) mm, rotated rx -180 ry 0 rz 134.32 deg; joints [58.889, -26.921, 122.809, 59.023, 86.961, 84.954, -584.321]
  MoveL 325 to (-48.58, 221.03, 50) mm, rotated rx 180 ry 0 rz 128.74 deg; joints [59.311, -26.978, 123.194, 59.459, 86.832, 84.649, -578.737]
  MoveL 326 to (-51.63, 225.99, 40) mm, rotated rx -180 ry 0 rz 123.38 deg; joints [59.736, -27.035, 123.574, 59.899, 86.709, 84.345, -573.376]
  MoveL 327 to (-54.06, 230.92, 30) mm, rotated rx -180 ry 0 rz 118.27 deg; joints [60.166, -27.089, 123.948, 60.343, 86.594, 84.042, -568.272]
  MoveL 328 to (-55.91, 235.73, 20) mm, rotated rx -180 ry 0 rz 113.46 deg; joints [60.599, -27.14, 124.316, 60.791, 86.484, 83.74, -563.465]
  MoveL 329 to (-57.23, 240.3, 10) mm, rotated rx -180 ry 0 rz 108.99 deg; joints [61.035, -27.188, 124.678, 61.243, 86.381, 83.438, -558.992]
  MoveL 330 to (-58.12, 244.54, 0) mm, rotated rx -180 ry 0 rz 104.89 deg; joints [61.476, -27.232, 125.032, 61.699, 86.284, 83.137, -554.894]
  MoveL 331 to (58.22, 245.2, 290) mm, rotated rx 180 ry 0 rz -104.27 deg; joints [50.189, -25.701, 112.829, 50.224, 91.839, 92.207, -705.735]
  Set speed (60.0 mm/s)
  MoveL 332 to (78.63, 249.2, 290) mm, rotated rx -180 ry 0 rz -97.82 deg; joints [50.189, -24.402, 112.105, 50.211, 91.47, 91.765, -712.181]
  MoveL 333 to (-58.12, 244.54, 0) mm, rotated rx -180 ry 0 rz 104.89 deg; joints [61.476, -27.232, 125.032, 61.699, 86.284, 83.137, -554.894]
  Set speed (60.0 mm/s)
  MoveL 334 to (-76.17, 234.21, 0) mm, rotated rx -180 ry 0 rz 108.7 deg; joints [61.476, -25.73, 124.214, 61.74, 85.96, 82.533, -558.703]
  MoveL 335 to (-58.12, 244.54, 0) mm, rotated rx -180 ry 0 rz 104.89 deg; joints [61.476, -27.232, 125.032, 61.699, 86.284, 83.137, -554.894]
  Set speed (60.0 mm/s)
  MoveL 336 to (-57.23, 240.3, 10) mm, rotated rx -180 ry 0 rz 108.99 deg; joints [61.035, -27.188, 124.678, 61.243, 86.381, 83.438, -558.992]
  MoveL 337 to (-55.91, 235.73, 20) mm, rotated rx -180 ry 0 rz 113.46 deg; joints [60.599, -27.14, 124.316, 60.791, 86.484, 83.74, -563.465]
  MoveL 338 to (-54.06, 230.92, 30) mm, rotated rx 180 ry 0 rz 118.27 deg; joints [60.166, -27.089, 123.948, 60.343, 86.594, 84.042, -568.272]
  MoveL 339 to (-51.63, 225.99, 40) mm, rotated rx -180 ry 0 rz 123.38 deg; joints [59.736, -27.035, 123.574, 59.899, 86.709, 84.345, -573.376]
  MoveL 340 to (-48.58, 221.03, 50) mm, rotated rx 180 ry 0 rz 128.74 deg; joints [59.311, -26.978, 123.194, 59.459, 86.832, 84.649, -578.737]
  MoveL 341 to (-44.86, 216.19, 60) mm, rotated rx -180 ry 0 rz 134.32 deg; joints [58.889, -26.921, 122.809, 59.023, 86.961, 84.954, -584.321]
  MoveL 342 to (-40.49, 211.59, 70) mm, rotated rx -180 ry 0 rz 140.09 deg; joints [58.471, -26.863, 122.42, 58.591, 87.097, 85.259, -590.093]
  MoveL 343 to (-35.48, 207.36, 80) mm, rotated rx -180 ry 0 rz 146.02 deg; joints [58.056, -26.805, 122.025, 58.163, 87.241, 85.567, -596.02]
  MoveL 344 to (-29.89, 203.62, 90) mm, rotated rx -180 ry 0 rz 152.07 deg; joints [57.646, -26.747, 121.627, 57.74, 87.391, 85.875, -602.072]
  MoveL 345 to (-23.78, 200.49, 100) mm, rotated rx -180 ry 0 rz 158.22 deg; joints [57.239, -26.692, 121.225, 57.32, 87.549, 86.185, -608.22]
  MoveL 346 to (-17.25, 198.06, 110) mm, rotated rx -180 ry 0 rz 164.44 deg; joints [56.835, -26.638, 120.82, 56.905, 87.714, 86.497, -614.435]
  MoveL 347 to (-10.42, 196.41, 120) mm, rotated rx -180 ry 0 rz 170.69 deg; joints [56.436, -26.586, 120.411, 56.495, 87.886, 86.811, -620.691]
  MoveL 348 to (-3.42, 195.58, 130) mm, rotated rx -180 ry 0 rz 176.96 deg; joints [56.04, -26.536, 120, 56.088, 88.066, 87.126, -626.961]
  MoveL 349 to (3.62, 195.59, 140) mm, rotated rx -180 ry 0 rz -176.78 deg; joints [55.647, -26.489, 119.585, 55.686, 88.254, 87.443, -633.219]
  MoveL 350 to (10.57, 196.44, 150) mm, rotated rx -180 ry 0 rz -170.56 deg; joints [55.259, -26.444, 119.167, 55.289, 88.449, 87.762, -639.438]
  MoveL 351 to (17.28, 198.07, 160) mm, rotated rx 180 ry 0 rz -164.41 deg; joints [54.874, -26.401, 118.747, 54.896, 88.651, 88.081, -645.594]
  MoveL 352 to (23.65, 200.44, 170) mm, rotated rx -180 ry 0 rz -158.34 deg; joints [54.492, -26.359, 118.322, 54.508, 88.86, 88.402, -651.658]
  MoveL 353 to (29.57, 203.44, 180) mm, rotated rx 180 ry 0 rz -152.4 deg; joints [54.114, -26.318, 117.894, 54.125, 89.076, 88.723, -657.602]
  MoveL 354 to (34.96, 206.97, 190) mm, rotated rx 180 ry 0 rz -146.6 deg; joints [53.74, -26.277, 117.462, 53.746, 89.299, 89.044, -663.399]
  MoveL 355 to (39.77, 210.92, 200) mm, rotated rx 180 ry 0 rz -140.98 deg; joints [53.369, -26.235, 117.026, 53.372, 89.528, 89.366, -669.016]
  MoveL 356 to (43.95, 215.15, 210) mm, rotated rx -180 ry 0 rz -135.58 deg; joints [53.002, -26.192, 116.584, 53.003, 89.764, 89.687, -674.422]
  MoveL 357 to (47.51, 219.54, 220) mm, rotated rx -180 ry 0 rz -130.42 deg; joints [52.638, -26.147, 116.138, 52.638, 90.005, 90.007, -679.584]
  MoveL 358 to (50.46, 223.96, 230) mm, rotated rx -180 ry 0 rz -125.53 deg; joints [52.278, -26.098, 115.685, 52.279, 90.253, 90.326, -684.466]
  MoveL 359 to (52.84, 228.29, 240) mm, rotated rx 180 ry 0 rz -120.97 deg; joints [51.921, -26.046, 115.227, 51.924, 90.505, 90.645, -689.031]
  MoveL 360 to (54.69, 232.42, 250) mm, rotated rx -180 ry 0 rz -116.76 deg; joints [51.568, -25.988, 114.762, 51.574, 90.763, 90.961, -693.242]
  MoveL 361 to (56.08, 236.26, 260) mm, rotated rx -180 ry 0 rz -112.94 deg; joints [51.218, -25.926, 114.289, 51.23, 91.025, 91.276, -697.057]
  MoveL 362 to (57.08, 239.72, 270) mm, rotated rx -180 ry 0 rz -109.56 deg; joints [50.872, -25.858, 113.81, 50.89, 91.292, 91.588, -700.439]
  MoveL 363 to (57.77, 242.72, 280) mm, rotated rx -180 ry 0 rz -106.66 deg; joints [50.529, -25.783, 113.323, 50.554, 91.563, 91.899, -703.345]
  MoveL 364 to (58.22, 245.2, 290) mm, rotated rx 180 ry 0 rz -104.27 deg; joints [50.189, -25.701, 112.829, 50.224, 91.839, 92.207, -705.735]
  MoveL 365 to (78.63, 249.2, 290) mm, rotated rx -180 ry 0 rz -97.82 deg; joints [50.189, -24.402, 112.105, 50.211, 91.47, 91.765, -712.181]
  Set speed (60.0 mm/s)
  MoveL 366 to (78.34, 245.85, 280) mm, rotated rx -180 ry 0 rz -100.24 deg; joints [50.529, -24.478, 112.597, 50.544, 91.195, 91.452, -709.758]
  MoveL 367 to (77.78, 241.77, 270) mm, rotated rx -180 ry 0 rz -103.19 deg; joints [50.872, -24.548, 113.082, 50.881, 90.925, 91.137, -706.809]
  MoveL 368 to (76.86, 237.05, 260) mm, rotated rx -180 ry 0 rz -106.63 deg; joints [51.218, -24.611, 113.559, 51.223, 90.659, 90.82, -703.374]
  MoveL 369 to (75.48, 231.77, 250) mm, rotated rx 180 ry 0 rz -110.51 deg; joints [51.568, -24.667, 114.028, 51.57, 90.397, 90.501, -699.493]
  MoveL 370 to (73.51, 226.04, 240) mm, rotated rx -180 ry 0 rz -114.79 deg; joints [51.921, -24.719, 114.49, 51.922, 90.141, 90.18, -695.208]
  MoveL 371 to (70.88, 219.99, 230) mm, rotated rx -180 ry 0 rz -119.44 deg; joints [52.278, -24.765, 114.946, 52.278, 89.889, 89.857, -690.555]
  MoveL 372 to (67.49, 213.75, 220) mm, rotated rx -180 ry 0 rz -124.42 deg; joints [52.638, -24.807, 115.395, 52.64, 89.643, 89.533, -685.575]
  MoveL 373 to (63.28, 207.47, 210) mm, rotated rx -180 ry 0 rz -129.69 deg; joints [53.002, -24.845, 115.838, 53.006, 89.403, 89.207, -680.305]
  MoveL 374 to (58.22, 201.33, 200) mm, rotated rx -180 ry 0 rz -135.22 deg; joints [53.369, -24.881, 116.275, 53.377, 89.168, 88.881, -674.781]
  MoveL 375 to (52.31, 195.49, 190) mm, rotated rx 180 ry 0 rz -140.96 deg; joints [53.74, -24.915, 116.708, 53.753, 88.94, 88.554, -669.037]
  MoveL 376 to (45.56, 190.13, 180) mm, rotated rx -180 ry 0 rz -146.89 deg; joints [54.114, -24.948, 117.136, 54.134, 88.718, 88.227, -663.107]
  MoveL 377 to (38.04, 185.42, 170) mm, rotated rx -180 ry 0 rz -152.98 deg; joints [54.492, -24.981, 117.559, 54.52, 88.503, 87.901, -657.024]
  MoveL 378 to (29.85, 181.5, 160) mm, rotated rx -180 ry 0 rz -159.18 deg; joints [54.874, -25.014, 117.979, 54.91, 88.295, 87.574, -650.818]
  MoveL 379 to (21.11, 178.51, 150) mm, rotated rx -180 ry 0 rz -165.48 deg; joints [55.259, -25.049, 118.396, 55.304, 88.094, 87.249, -644.519]
  MoveL 380 to (11.96, 176.54, 140) mm, rotated rx -180 ry 0 rz -171.84 deg; joints [55.647, -25.085, 118.809, 55.704, 87.9, 86.925, -638.157]
  MoveL 381 to (2.59, 175.67, 130) mm, rotated rx -180 ry 0 rz -178.24 deg; joints [56.04, -25.124, 119.219, 56.108, 87.714, 86.602, -631.758]
  MoveL 382 to (-6.83, 175.92, 120) mm, rotated rx -180 ry 0 rz 175.35 deg; joints [56.436, -25.165, 119.627, 56.516, 87.535, 86.28, -625.352]
  MoveL 383 to (-16.13, 177.3, 110) mm, rotated rx -180 ry 0 rz 168.97 deg; joints [56.835, -25.208, 120.031, 56.928, 87.364, 85.96, -618.967]
  MoveL 384 to (-25.11, 179.73, 100) mm, rotated rx 180 ry 0 rz 162.63 deg; joints [57.239, -25.254, 120.433, 57.345, 87.2, 85.642, -612.629]
  MoveL 385 to (-33.62, 183.16, 90) mm, rotated rx -180 ry 0 rz 156.37 deg; joints [57.646, -25.302, 120.831, 57.766, 87.044, 85.325, -606.369]
  MoveL 386 to (-41.52, 187.45, 80) mm, rotated rx -180 ry 0 rz 150.21 deg; joints [58.056, -25.352, 121.226, 58.192, 86.896, 85.01, -600.214]
  MoveL 387 to (-48.7, 192.48, 70) mm, rotated rx -180 ry 0 rz 144.2 deg; joints [58.471, -25.402, 121.617, 58.621, 86.755, 84.697, -594.197]
  MoveL 388 to (-55.08, 198.08, 60) mm, rotated rx -180 ry 0 rz 138.35 deg; joints [58.889, -25.453, 122.005, 59.055, 86.62, 84.385, -588.347]
  MoveL 389 to (-60.61, 204.07, 50) mm, rotated rx -180 ry 0 rz 132.7 deg; joints [59.311, -25.504, 122.387, 59.492, 86.494, 84.074, -582.698]
  MoveL 390 to (-65.29, 210.3, 40) mm, rotated rx 180 ry 0 rz 127.28 deg; joints [59.736, -25.554, 122.764, 59.934, 86.373, 83.764, -577.284]
  MoveL 391 to (-69.12, 216.58, 30) mm, rotated rx -180 ry 0 rz 122.14 deg; joints [60.166, -25.603, 123.136, 60.38, 86.26, 83.455, -572.14]
  MoveL 392 to (-72.16, 222.75, 20) mm, rotated rx -180 ry 0 rz 117.3 deg; joints [60.599, -25.648, 123.502, 60.829, 86.154, 83.147, -567.303]
  MoveL 393 to (-74.48, 228.68, 10) mm, rotated rx 180 ry 0 rz 112.81 deg; joints [61.035, -25.691, 123.862, 61.282, 86.053, 82.84, -562.811]
  MoveL 394 to (-76.17, 234.21, 0) mm, rotated rx -180 ry 0 rz 108.7 deg; joints [61.476, -25.73, 124.214, 61.74, 85.96, 82.533, -558.703]
  MoveL 395 to (78.63, 249.2, 290) mm, rotated rx -180 ry 0 rz -97.82 deg; joints [50.189, -24.402, 112.105, 50.211, 91.47, 91.765, -712.181]
  Set speed (60.0 mm/s)
  MoveL 396 to (58.93, 255.88, 290) mm, rotated rx -180 ry 0 rz -94 deg; joints [50.189, -25.769, 112.866, 50.225, 91.858, 92.231, -715.998]
  MoveL 397 to (-76.17, 234.21, 0) mm, rotated rx -180 ry 0 rz 108.7 deg; joints [61.476, -25.73, 124.214, 61.74, 85.96, 82.533, -558.703]
  Set speed (60.0 mm/s)
  MoveL 398 to (-55.37, 234.2, 0) mm, rotated rx 180 ry 0 rz 114.99 deg; joints [61.476, -27.161, 124.995, 61.701, 86.268, 83.108, -564.986]
  MoveL 399 to (-76.17, 234.21, 0) mm, rotated rx 180 ry 0 rz 108.7 deg; joints [61.476, -25.73, 124.214, 61.74, 85.96, 82.533, -558.703]
  Set speed (60.0 mm/s)
  MoveL 400 to (-74.48, 228.68, 10) mm, rotated rx 180 ry 0 rz 112.81 deg; joints [61.035, -25.691, 123.862, 61.282, 86.053, 82.84, -562.811]
  MoveL 401 to (-72.16, 222.75, 20) mm, rotated rx -180 ry 0 rz 117.3 deg; joints [60.599, -25.648, 123.502, 60.829, 86.154, 83.147, -567.303]
  MoveL 402 to (-69.12, 216.58, 30) mm, rotated rx -180 ry 0 rz 122.14 deg; joints [60.166, -25.603, 123.136, 60.38, 86.26, 83.455, -572.14]
  MoveL 403 to (-65.29, 210.3, 40) mm, rotated rx 180 ry 0 rz 127.28 deg; joints [59.736, -25.554, 122.764, 59.934, 86.373, 83.764, -577.284]
  MoveL 404 to (-60.61, 204.07, 50) mm, rotated rx -180 ry 0 rz 132.7 deg; joints [59.311, -25.504, 122.387, 59.492, 86.494, 84.074, -582.698]
  MoveL 405 to (-55.08, 198.08, 60) mm, rotated rx -180 ry 0 rz 138.35 deg; joints [58.889, -25.453, 122.005, 59.055, 86.62, 84.385, -588.347]
  MoveL 406 to (-48.7, 192.48, 70) mm, rotated rx -180 ry 0 rz 144.2 deg; joints [58.471, -25.402, 121.617, 58.621, 86.755, 84.697, -594.197]
  MoveL 407 to (-41.52, 187.45, 80) mm, rotated rx -180 ry 0 rz 150.21 deg; joints [58.056, -25.352, 121.226, 58.192, 86.896, 85.01, -600.214]
  MoveL 408 to (-33.62, 183.16, 90) mm, rotated rx -180 ry 0 rz 156.37 deg; joints [57.646, -25.302, 120.831, 57.766, 87.044, 85.325, -606.369]
  MoveL 409 to (-25.11, 179.73, 100) mm, rotated rx 180 ry 0 rz 162.63 deg; joints [57.239, -25.254, 120.433, 57.345, 87.2, 85.642, -612.629]
  MoveL 410 to (-16.13, 177.3, 110) mm, rotated rx -180 ry 0 rz 168.97 deg; joints [56.835, -25.208, 120.031, 56.928, 87.364, 85.96, -618.967]
  MoveL 411 to (-6.83, 175.92, 120) mm, rotated rx -180 ry 0 rz 175.35 deg; joints [56.436, -25.165, 119.627, 56.516, 87.535, 86.28, -625.352]
  MoveL 412 to (2.59, 175.67, 130) mm, rotated rx -180 ry 0 rz -178.24 deg; joints [56.04, -25.124, 119.219, 56.108, 87.714, 86.602, -631.758]
  MoveL 413 to (11.96, 176.54, 140) mm, rotated rx -180 ry 0 rz -171.84 deg; joints [55.647, -25.085, 118.809, 55.704, 87.9, 86.925, -638.157]
  MoveL 414 to (21.11, 178.51, 150) mm, rotated rx -180 ry 0 rz -165.48 deg; joints [55.259, -25.049, 118.396, 55.304, 88.094, 87.249, -644.519]
  MoveL 415 to (29.85, 181.5, 160) mm, rotated rx -180 ry 0 rz -159.18 deg; joints [54.874, -25.014, 117.979, 54.91, 88.295, 87.574, -650.818]
  MoveL 416 to (38.04, 185.42, 170) mm, rotated rx -180 ry 0 rz -152.98 deg; joints [54.492, -24.981, 117.559, 54.52, 88.503, 87.901, -657.024]
  MoveL 417 to (45.56, 190.13, 180) mm, rotated rx -180 ry 0 rz -146.89 deg; joints [54.114, -24.948, 117.136, 54.134, 88.718, 88.227, -663.107]
  MoveL 418 to (52.31, 195.49, 190) mm, rotated rx -180 ry 0 rz -140.96 deg; joints [53.74, -24.915, 116.708, 53.753, 88.94, 88.554, -669.037]
  MoveL 419 to (58.22, 201.33, 200) mm, rotated rx -180 ry 0 rz -135.22 deg; joints [53.369, -24.881, 116.275, 53.377, 89.168, 88.881, -674.781]
  MoveL 420 to (63.28, 207.47, 210) mm, rotated rx -180 ry 0 rz -129.69 deg; joints [53.002, -24.845, 115.838, 53.006, 89.403, 89.207, -680.305]
  MoveL 421 to (67.49, 213.75, 220) mm, rotated rx -180 ry 0 rz -124.42 deg; joints [52.638, -24.807, 115.395, 52.64, 89.643, 89.533, -685.575]
  MoveL 422 to (70.88, 219.99, 230) mm, rotated rx -180 ry 0 rz -119.44 deg; joints [52.278, -24.765, 114.946, 52.278, 89.889, 89.857, -690.555]
  MoveL 423 to (73.51, 226.04, 240) mm, rotated rx -180 ry 0 rz -114.79 deg; joints [51.921, -24.719, 114.49, 51.922, 90.141, 90.18, -695.208]
  MoveL 424 to (75.48, 231.77, 250) mm, rotated rx 180 ry 0 rz -110.51 deg; joints [51.568, -24.667, 114.028, 51.57, 90.397, 90.501, -699.493]
  MoveL 425 to (76.86, 237.05, 260) mm, rotated rx -180 ry 0 rz -106.63 deg; joints [51.218, -24.611, 113.559, 51.223, 90.659, 90.82, -703.374]
  MoveL 426 to (77.78, 241.77, 270) mm, rotated rx -180 ry 0 rz -103.19 deg; joints [50.872, -24.548, 113.082, 50.881, 90.925, 91.137, -706.809]
  MoveL 427 to (78.34, 245.85, 280) mm, rotated rx 180 ry 0 rz -100.24 deg; joints [50.529, -24.478, 112.597, 50.544, 91.195, 91.452, -709.758]
  MoveL 428 to (78.63, 249.2, 290) mm, rotated rx -180 ry 0 rz -97.82 deg; joints [50.189, -24.402, 112.105, 50.211, 91.47, 91.765, -712.181]
  MoveL 429 to (58.93, 255.88, 290) mm, rotated rx -180 ry 0 rz -94 deg; joints [50.189, -25.769, 112.866, 50.225, 91.858, 92.231, -715.998]
  Set speed (60.0 mm/s)
  MoveL 430 to (58.94, 253.36, 280) mm, rotated rx -180 ry 0 rz -96.43 deg; joints [50.529, -25.85, 113.36, 50.555, 91.583, 91.923, -713.568]
  MoveL 431 to (58.8, 250.28, 270) mm, rotated rx -180 ry 0 rz -99.38 deg; joints [50.872, -25.924, 113.846, 50.89, 91.311, 91.612, -710.615]
  MoveL 432 to (58.44, 246.7, 260) mm, rotated rx 180 ry 0 rz -102.82 deg; joints [51.218, -25.991, 114.325, 51.23, 91.044, 91.299, -707.181]
  MoveL 433 to (57.77, 242.68, 250) mm, rotated rx -180 ry 0 rz -106.69 deg; joints [51.568, -26.053, 114.796, 51.575, 90.781, 90.984, -703.306]
  MoveL 434 to (56.69, 238.28, 240) mm, rotated rx -180 ry 0 rz -110.97 deg; joints [51.921, -26.108, 115.261, 51.924, 90.523, 90.667, -699.034]
  MoveL 435 to (55.14, 233.59, 230) mm, rotated rx -180 ry 0 rz -115.59 deg; joints [52.278, -26.158, 115.718, 52.279, 90.269, 90.348, -694.405]
  MoveL 436 to (53.04, 228.71, 220) mm, rotated rx -180 ry 0 rz -120.54 deg; joints [52.638, -26.204, 116.169, 52.638, 90.021, 90.028, -689.46]
  MoveL 437 to (50.33, 223.75, 210) mm, rotated rx -180 ry 0 rz -125.76 deg; joints [53.002, -26.245, 116.613, 53.003, 89.779, 89.706, -684.235]
  MoveL 438 to (46.98, 218.83, 200) mm, rotated rx -180 ry 0 rz -131.23 deg; joints [53.369, -26.284, 117.052, 53.372, 89.542, 89.384, -678.769]
  MoveL 439 to (42.97, 214.08, 190) mm, rotated rx -180 ry 0 rz -136.9 deg; joints [53.74, -26.321, 117.486, 53.746, 89.311, 89.06, -673.096]
  MoveL 440 to (38.31, 209.62, 180) mm, rotated rx -180 ry 0 rz -142.75 deg; joints [54.114, -26.356, 117.915, 54.124, 89.086, 88.737, -667.251]
  MoveL 441 to (33.03, 205.6, 170) mm, rotated rx 180 ry 0 rz -148.74 deg; joints [54.492, -26.391, 118.34, 54.508, 88.868, 88.413, -661.263]
  MoveL 442 to (27.19, 202.13, 160) mm, rotated rx 180 ry 0 rz -154.84 deg; joints [54.874, -26.426, 118.76, 54.896, 88.657, 88.09, -655.164]
  MoveL 443 to (20.88, 199.3, 150) mm, rotated rx 180 ry 0 rz -161.02 deg; joints [55.259, -26.462, 119.177, 55.289, 88.453, 87.768, -648.983]
  MoveL 444 to (14.2, 197.22, 140) mm, rotated rx -180 ry 0 rz -167.25 deg; joints [55.647, -26.499, 119.59, 55.686, 88.256, 87.447, -642.746]
  MoveL 445 to (7.28, 195.93, 130) mm, rotated rx 180 ry 0 rz -173.52 deg; joints [56.04, -26.539, 120.001, 56.088, 88.067, 87.127, -636.481]
  MoveL 446 to (0.24, 195.48, 120) mm, rotated rx 180 ry 0 rz -179.79 deg; joints [56.436, -26.58, 120.408, 56.495, 87.885, 86.809, -630.213]
  MoveL 447 to (-6.77, 195.87, 110) mm, rotated rx 180 ry 0 rz 173.97 deg; joints [56.835, -26.624, 120.812, 56.906, 87.71, 86.492, -623.969]
  MoveL 448 to (-13.63, 197.08, 100) mm, rotated rx 180 ry 0 rz 167.78 deg; joints [57.239, -26.67, 121.214, 57.321, 87.543, 86.177, -617.775]
  MoveL 449 to (-20.21, 199.05, 90) mm, rotated rx -180 ry 0 rz 161.66 deg; joints [57.646, -26.719, 121.611, 57.74, 87.384, 85.864, -611.658]
  MoveL 450 to (-26.38, 201.72, 80) mm, rotated rx -180 ry 0 rz 155.64 deg; joints [58.056, -26.769, 122.006, 58.164, 87.232, 85.553, -605.644]
  MoveL 451 to (-32.08, 204.97, 70) mm, rotated rx -180 ry 0 rz 149.76 deg; joints [58.471, -26.82, 122.397, 58.592, 87.087, 85.243, -599.763]
  MoveL 452 to (-37.21, 208.71, 60) mm, rotated rx -180 ry 0 rz 144.04 deg; joints [58.889, -26.873, 122.784, 59.024, 86.95, 84.934, -594.043]
  MoveL 453 to (-41.73, 212.8, 50) mm, rotated rx -180 ry 0 rz 138.52 deg; joints [59.311, -26.925, 123.166, 59.46, 86.819, 84.628, -588.517]
  MoveL 454 to (-45.64, 217.12, 40) mm, rotated rx -180 ry 0 rz 133.22 deg; joints [59.736, -26.976, 123.543, 59.9, 86.696, 84.322, -583.217]
  MoveL 455 to (-48.92, 221.54, 30) mm, rotated rx -180 ry 0 rz 128.18 deg; joints [60.166, -27.027, 123.915, 60.345, 86.579, 84.017, -578.176]
  MoveL 456 to (-51.6, 225.93, 20) mm, rotated rx -180 ry 0 rz 123.43 deg; joints [60.599, -27.075, 124.281, 60.793, 86.469, 83.713, -573.433]
  MoveL 457 to (-53.73, 230.19, 10) mm, rotated rx -180 ry 0 rz 119.02 deg; joints [61.035, -27.12, 124.641, 61.245, 86.366, 83.41, -569.023]
  MoveL 458 to (-55.37, 234.2, 0) mm, rotated rx -180 ry 0 rz 114.99 deg; joints [61.476, -27.161, 124.995, 61.701, 86.268, 83.108, -564.986]
  MoveL 459 to (58.93, 255.88, 290) mm, rotated rx -180 ry 0 rz -94 deg; joints [50.189, -25.769, 112.866, 50.225, 91.858, 92.231, -715.998]
  Set speed (60.0 mm/s)
  MoveL 460 to (37.11, 300.24, 290) mm, rotated rx -180 ry 0 rz -42.69 deg; joints [50.189, -26.061, 113.024, 50.228, 91.944, 92.334, -767.315]
  MoveL 461 to (-55.37, 234.2, 0) mm, rotated rx -180 ry 0 rz 114.99 deg; joints [61.476, -27.161, 124.995, 61.701, 86.268, 83.108, -924.986]
  Set speed (60.0 mm/s)
  MoveL 462 to (-20.49, 199.16, 0) mm, rotated rx -180 ry 0 rz 161.39 deg; joints [61.476, -26.93, 124.871, 61.707, 86.217, 83.013, -971.385]
  MoveL 463 to (-55.37, 234.2, 0) mm, rotated rx -180 ry 0 rz 114.99 deg; joints [61.476, -27.161, 124.995, 61.701, 86.268, 83.108, -924.986]
  Set speed (60.0 mm/s)
  MoveL 464 to (-53.73, 230.19, 10) mm, rotated rx -180 ry 0 rz 119.02 deg; joints [61.035, -27.12, 124.641, 61.245, 86.366, 83.41, -929.023]
  MoveL 465 to (-51.6, 225.93, 20) mm, rotated rx -180 ry 0 rz 123.43 deg; joints [60.599, -27.075, 124.281, 60.793, 86.469, 83.713, -933.433]
  MoveL 466 to (-48.92, 221.54, 30) mm, rotated rx -180 ry 0 rz 128.18 deg; joints [60.166, -27.027, 123.915, 60.345, 86.579, 84.017, -938.176]
  MoveL 467 to (-45.64, 217.12, 40) mm, rotated rx -180 ry 0 rz 133.22 deg; joints [59.736, -26.976, 123.543, 59.9, 86.696, 84.322, -943.217]
  MoveL 468 to (-41.73, 212.8, 50) mm, rotated rx -180 ry 0 rz 138.52 deg; joints [59.311, -26.925, 123.166, 59.46, 86.819, 84.628, -948.517]
  MoveL 469 to (-37.21, 208.71, 60) mm, rotated rx -180 ry 0 rz 144.04 deg; joints [58.889, -26.873, 122.784, 59.024, 86.95, 84.934, -954.043]
  MoveL 470 to (-32.08, 204.97, 70) mm, rotated rx 180 ry 0 rz 149.76 deg; joints [58.471, -26.82, 122.397, 58.592, 87.087, 85.243, -959.763]
  MoveL 471 to (-26.38, 201.72, 80) mm, rotated rx -180 ry 0 rz 155.64 deg; joints [58.056, -26.769, 122.006, 58.164, 87.232, 85.553, -965.644]
  MoveL 472 to (-20.21, 199.05, 90) mm, rotated rx -180 ry 0 rz 161.66 deg; joints [57.646, -26.719, 121.611, 57.74, 87.384, 85.864, -971.658]
  MoveL 473 to (-13.63, 197.08, 100) mm, rotated rx 180 ry 0 rz 167.78 deg; joints [57.239, -26.67, 121.214, 57.321, 87.543, 86.177, -977.775]
  MoveL 474 to (-6.77, 195.87, 110) mm, rotated rx -180 ry 0 rz 173.97 deg; joints [56.835, -26.624, 120.812, 56.906, 87.71, 86.492, -983.969]
  MoveL 475 to (0.24, 195.48, 120) mm, rotated rx -180 ry 0 rz -179.79 deg; joints [56.436, -26.58, 120.408, 56.495, 87.885, 86.809, -990.213]
  MoveL 476 to (7.28, 195.93, 130) mm, rotated rx -180 ry 0 rz -173.52 deg; joints [56.04, -26.539, 120.001, 56.088, 88.067, 87.127, -996.481]
  MoveL 477 to (14.2, 197.22, 140) mm, rotated rx -180 ry 0 rz -167.25 deg; joints [55.647, -26.499, 119.59, 55.686, 88.256, 87.447, -1002.746]
  MoveL 478 to (20.88, 199.3, 150) mm, rotated rx 180 ry 0 rz -161.02 deg; joints [55.259, -26.462, 119.177, 55.289, 88.453, 87.768, -1008.983]
  MoveL 479 to (27.19, 202.13, 160) mm, rotated rx -180 ry 0 rz -154.84 deg; joints [54.874, -26.426, 118.76, 54.896, 88.657, 88.09, -1015.164]
  MoveL 480 to (33.03, 205.6, 170) mm, rotated rx -180 ry 0 rz -148.74 deg; joints [54.492, -26.391, 118.34, 54.508, 88.868, 88.413, -1021.263]
  MoveL 481 to (38.31, 209.62, 180) mm, rotated rx -180 ry 0 rz -142.75 deg; joints [54.114, -26.356, 117.915, 54.124, 89.086, 88.737, -1027.251]
  MoveL 482 to (42.97, 214.08, 190) mm, rotated rx -180 ry 0 rz -136.9 deg; joints [53.74, -26.321, 117.486, 53.746, 89.311, 89.06, -1033.096]
  MoveL 483 to (46.98, 218.83, 200) mm, rotated rx 180 ry 0 rz -131.23 deg; joints [53.369, -26.284, 117.052, 53.372, 89.542, 89.384, -1038.769]
  MoveL 484 to (50.33, 223.75, 210) mm, rotated rx -180 ry 0 rz -125.76 deg; joints [53.002, -26.245, 116.613, 53.003, 89.779, 89.706, -1044.235]
  MoveL 485 to (53.04, 228.71, 220) mm, rotated rx -180 ry 0 rz -120.54 deg; joints [52.638, -26.204, 116.169, 52.638, 90.021, 90.028, -1049.46]
  MoveL 486 to (55.14, 233.59, 230) mm, rotated rx -180 ry 0 rz -115.59 deg; joints [52.278, -26.158, 115.718, 52.279, 90.269, 90.348, -1054.405]
  MoveL 487 to (56.69, 238.28, 240) mm, rotated rx -180 ry 0 rz -110.97 deg; joints [51.921, -26.108, 115.261, 51.924, 90.523, 90.667, -1059.034]
  MoveL 488 to (57.77, 242.68, 250) mm, rotated rx -180 ry 0 rz -106.69 deg; joints [51.568, -26.053, 114.796, 51.575, 90.781, 90.984, -1063.306]
  MoveL 489 to (58.44, 246.7, 260) mm, rotated rx -180 ry 0 rz -102.82 deg; joints [51.218, -25.991, 114.325, 51.23, 91.044, 91.299, -1067.181]
  MoveL 490 to (58.8, 250.28, 270) mm, rotated rx 180 ry 0 rz -99.38 deg; joints [50.872, -25.924, 113.846, 50.89, 91.311, 91.612, -1070.615]
  MoveL 491 to (58.94, 253.36, 280) mm, rotated rx -180 ry 0 rz -96.43 deg; joints [50.529, -25.85, 113.36, 50.555, 91.583, 91.923, -1073.568]
  MoveL 492 to (58.93, 255.88, 290) mm, rotated rx -180 ry 0 rz -94 deg; joints [50.189, -25.769, 112.866, 50.225, 91.858, 92.231, -1075.998]
  MoveL 493 to (37.11, 300.24, 290) mm, rotated rx -180 ry 0 rz -42.69 deg; joints [50.189, -26.061, 113.024, 50.228, 91.944, 92.334, -1127.315]
  Set speed (60.0 mm/s)
  MoveL 494 to (39.03, 298.61, 280) mm, rotated rx -180 ry 0 rz -45.31 deg; joints [50.529, -26.148, 113.522, 50.558, 91.669, 92.028, -1124.686]
  MoveL 495 to (41.29, 296.51, 270) mm, rotated rx 180 ry 0 rz -48.51 deg; joints [50.872, -26.229, 114.011, 50.893, 91.399, 91.72, -1121.487]
  MoveL 496 to (43.78, 293.91, 260) mm, rotated rx -180 ry 0 rz -52.23 deg; joints [51.218, -26.302, 114.493, 51.232, 91.133, 91.41, -1117.765]
  MoveL 497 to (46.4, 290.79, 250) mm, rotated rx -180 ry 0 rz -56.43 deg; joints [51.568, -26.368, 114.967, 51.576, 90.871, 91.098, -1113.565]
  MoveL 498 to (49.06, 287.12, 240) mm, rotated rx -180 ry 0 rz -61.06 deg; joints [51.921, -26.427, 115.433, 51.925, 90.613, 90.783, -1108.935]
  MoveL 499 to (51.62, 282.9, 230) mm, rotated rx -180 ry 0 rz -66.08 deg; joints [52.278, -26.479, 115.891, 52.28, 90.36, 90.465, -1103.922]
  MoveL 500 to (53.98, 278.14, 220) mm, rotated rx 180 ry 0 rz -71.43 deg; joints [52.638, -26.524, 116.342, 52.638, 90.111, 90.145, -1098.571]
  MoveL 501 to (56, 272.86, 210) mm, rotated rx 180 ry 0 rz -77.07 deg; joints [53.002, -26.563, 116.785, 53.002, 89.867, 89.823, -1092.931]
  MoveL 502 to (57.57, 267.12, 200) mm, rotated rx -180 ry 0 rz -82.95 deg; joints [53.369, -26.595, 117.22, 53.371, 89.627, 89.498, -1087.046]
  MoveL 503 to (58.59, 260.98, 190) mm, rotated rx -180 ry 0 rz -89.04 deg; joints [53.74, -26.621, 117.648, 53.744, 89.393, 89.172, -1080.96]
  MoveL 504 to (58.95, 254.55, 180) mm, rotated rx -180 ry 0 rz -95.29 deg; joints [54.114, -26.642, 118.069, 54.123, 89.163, 88.844, -1074.714]
  MoveL 505 to (58.59, 247.92, 170) mm, rotated rx 180 ry 0 rz -101.65 deg; joints [54.492, -26.659, 118.484, 54.506, 88.94, 88.514, -1068.348]
  MoveL 506 to (57.45, 241.22, 160) mm, rotated rx -180 ry 0 rz -108.1 deg; joints [54.874, -26.673, 118.893, 54.894, 88.723, 88.184, -1061.898]
  MoveL 507 to (55.51, 234.59, 150) mm, rotated rx -180 ry 0 rz -114.6 deg; joints [55.259, -26.684, 119.297, 55.287, 88.511, 87.852, -1055.4]
  MoveL 508 to (52.77, 228.15, 140) mm, rotated rx -180 ry 0 rz -121.12 deg; joints [55.647, -26.693, 119.695, 55.684, 88.307, 87.521, -1048.885]
  MoveL 509 to (49.26, 222.05, 130) mm, rotated rx 180 ry 0 rz -127.62 deg; joints [56.04, -26.702, 120.089, 56.086, 88.109, 87.19, -1042.384]
  MoveL 510 to (45.04, 216.4, 120) mm, rotated rx -180 ry 0 rz -134.07 deg; joints [56.436, -26.711, 120.479, 56.493, 87.918, 86.859, -1035.926]
  MoveL 511 to (40.19, 211.31, 110) mm, rotated rx -180 ry 0 rz -140.46 deg; joints [56.835, -26.721, 120.864, 56.904, 87.735, 86.53, -1029.537]
  MoveL 512 to (34.83, 206.87, 100) mm, rotated rx -180 ry 0 rz -146.76 deg; joints [57.239, -26.732, 121.247, 57.32, 87.559, 86.201, -1023.245]
  MoveL 513 to (29.06, 203.14, 90) mm, rotated rx -180 ry 0 rz -152.93 deg; joints [57.646, -26.744, 121.625, 57.74, 87.39, 85.874, -1017.074]
  MoveL 514 to (23.03, 200.17, 80) mm, rotated rx -180 ry 0 rz -158.95 deg; joints [58.056, -26.759, 122.001, 58.164, 87.23, 85.549, -1011.051]
  MoveL 515 to (16.86, 197.94, 70) mm, rotated rx -180 ry 0 rz -164.8 deg; joints [58.471, -26.776, 122.373, 58.593, 87.077, 85.225, -1005.201]
  MoveL 516 to (10.69, 196.46, 60) mm, rotated rx -180 ry 0 rz -170.45 deg; joints [58.889, -26.795, 122.742, 59.026, 86.931, 84.904, -999.549]
  MoveL 517 to (4.64, 195.67, 50) mm, rotated rx -180 ry 0 rz -175.88 deg; joints [59.311, -26.815, 123.107, 59.463, 86.794, 84.584, -994.124]
  MoveL 518 to (-1.18, 195.49, 40) mm, rotated rx -180 ry 0 rz 178.95 deg; joints [59.736, -26.837, 123.468, 59.904, 86.664, 84.266, -988.952]
  MoveL 519 to (-6.67, 195.86, 30) mm, rotated rx -180 ry 0 rz 174.06 deg; joints [60.166, -26.861, 123.826, 60.349, 86.541, 83.95, -984.062]
  MoveL 520 to (-11.76, 196.67, 20) mm, rotated rx -180 ry 0 rz 169.48 deg; joints [60.599, -26.884, 124.179, 60.797, 86.426, 83.636, -979.483]
  MoveL 521 to (-16.38, 197.8, 10) mm, rotated rx 180 ry 0 rz 165.25 deg; joints [61.035, -26.908, 124.528, 61.25, 86.318, 83.324, -975.247]
  MoveL 522 to (-20.49, 199.16, 0) mm, rotated rx 180 ry 0 rz 161.39 deg; joints [61.476, -26.93, 124.871, 61.707, 86.217, 83.013, -971.385]
  MoveL 523 to (37.11, 300.24, 290) mm, rotated rx -180 ry 0 rz -42.69 deg; joints [50.189, -26.061, 113.024, 50.228, 91.944, 92.334, -1127.315]
  Set speed (60.0 mm/s)
  MoveL 524 to (43.85, 319.91, 290) mm, rotated rx -180 ry 0 rz -36.2 deg; joints [50.189, -24.747, 112.3, 50.214, 91.566, 91.88, -1133.803]
  MoveL 525 to (-20.49, 199.16, 0) mm, rotated rx -180 ry 0 rz 161.39 deg; joints [61.476, -26.93, 124.871, 61.707, 86.217, 83.013, -971.385]
  Set speed (60.0 mm/s)
  MoveL 526 to (-20.57, 178.36, 0) mm, rotated rx -180 ry 0 rz 165.86 deg; joints [61.476, -25.451, 124.058, 61.747, 85.902, 82.424, -975.856]
  MoveL 527 to (-20.49, 199.16, 0) mm, rotated rx 180 ry 0 rz 161.39 deg; joints [61.476, -26.93, 124.871, 61.707, 86.217, 83.013, -971.385]
  Set speed (60.0 mm/s)
  MoveL 528 to (-16.38, 197.8, 10) mm, rotated rx -180 ry 0 rz 165.25 deg; joints [61.035, -26.908, 124.528, 61.25, 86.318, 83.324, -975.247]
  MoveL 529 to (-11.76, 196.67, 20) mm, rotated rx -180 ry 0 rz 169.48 deg; joints [60.599, -26.884, 124.179, 60.797, 86.426, 83.636, -979.483]
  MoveL 530 to (-6.67, 195.86, 30) mm, rotated rx -180 ry 0 rz 174.06 deg; joints [60.166, -26.861, 123.826, 60.349, 86.541, 83.95, -984.062]
  MoveL 531 to (-1.18, 195.49, 40) mm, rotated rx 180 ry 0 rz 178.95 deg; joints [59.736, -26.837, 123.468, 59.904, 86.664, 84.266, -988.952]
  MoveL 532 to (4.64, 195.67, 50) mm, rotated rx 180 ry 0 rz -175.88 deg; joints [59.311, -26.815, 123.107, 59.463, 86.794, 84.584, -994.124]
  MoveL 533 to (10.69, 196.46, 60) mm, rotated rx -180 ry 0 rz -170.45 deg; joints [58.889, -26.795, 122.742, 59.026, 86.931, 84.904, -999.549]
  MoveL 534 to (16.86, 197.94, 70) mm, rotated rx -180 ry 0 rz -164.8 deg; joints [58.471, -26.776, 122.373, 58.593, 87.077, 85.225, -1005.201]
  MoveL 535 to (23.03, 200.17, 80) mm, rotated rx -180 ry 0 rz -158.95 deg; joints [58.056, -26.759, 122.001, 58.164, 87.23, 85.549, -1011.051]
  MoveL 536 to (29.06, 203.14, 90) mm, rotated rx -180 ry 0 rz -152.93 deg; joints [57.646, -26.744, 121.625, 57.74, 87.39, 85.874, -1017.074]
  MoveL 537 to (34.83, 206.87, 100) mm, rotated rx -180 ry 0 rz -146.76 deg; joints [57.239, -26.732, 121.247, 57.32, 87.559, 86.201, -1023.245]
  MoveL 538 to (40.19, 211.31, 110) mm, rotated rx -180 ry 0 rz -140.46 deg; joints [56.835, -26.721, 120.864, 56.904, 87.735, 86.53, -1029.537]
  MoveL 539 to (45.04, 216.4, 120) mm, rotated rx 180 ry 0 rz -134.07 deg; joints [56.436, -26.711, 120.479, 56.493, 87.918, 86.859, -1035.926]
  MoveL 540 to (49.26, 222.05, 130) mm, rotated rx -180 ry 0 rz -127.62 deg; joints [56.04, -26.702, 120.089, 56.086, 88.109, 87.19, -1042.384]
  MoveL 541 to (52.77, 228.15, 140) mm, rotated rx -180 ry 0 rz -121.12 deg; joints [55.647, -26.693, 119.695, 55.684, 88.307, 87.521, -1048.885]
  MoveL 542 to (55.51, 234.59, 150) mm, rotated rx -180 ry 0 rz -114.6 deg; joints [55.259, -26.684, 119.297, 55.287, 88.511, 87.852, -1055.4]
  MoveL 543 to (57.45, 241.22, 160) mm, rotated rx 180 ry 0 rz -108.1 deg; joints [54.874, -26.673, 118.893, 54.894, 88.723, 88.184, -1061.898]
  MoveL 544 to (58.59, 247.92, 170) mm, rotated rx -180 ry 0 rz -101.65 deg; joints [54.492, -26.659, 118.484, 54.506, 88.94, 88.514, -1068.348]
  MoveL 545 to (58.95, 254.55, 180) mm, rotated rx -180 ry 0 rz -95.29 deg; joints [54.114, -26.642, 118.069, 54.123, 89.163, 88.844, -1074.714]
  MoveL 546 to (58.59, 260.98, 190) mm, rotated rx -180 ry 0 rz -89.04 deg; joints [53.74, -26.621, 117.648, 53.744, 89.393, 89.172, -1080.96]
  MoveL 547 to (57.57, 267.12, 200) mm, rotated rx -180 ry 0 rz -82.95 deg; joints [53.369, -26.595, 117.22, 53.371, 89.627, 89.498, -1087.046]
  MoveL 548 to (56, 272.86, 210) mm, rotated rx -180 ry 0 rz -77.07 deg; joints [53.002, -26.563, 116.785, 53.002, 89.867, 89.823, -1092.931]
  MoveL 549 to (53.98, 278.14, 220) mm, rotated rx -180 ry 0 rz -71.43 deg; joints [52.638, -26.524, 116.342, 52.638, 90.111, 90.145, -1098.571]
  MoveL 550 to (51.62, 282.9, 230) mm, rotated rx -180 ry 0 rz -66.08 deg; joints [52.278, -26.479, 115.891, 52.28, 90.36, 90.465, -1103.922]
  MoveL 551 to (49.06, 287.12, 240) mm, rotated rx -180 ry 0 rz -61.06 deg; joints [51.921, -26.427, 115.433, 51.925, 90.613, 90.783, -1108.935]
  MoveL 552 to (46.4, 290.79, 250) mm, rotated rx -180 ry 0 rz -56.43 deg; joints [51.568, -26.368, 114.967, 51.576, 90.871, 91.098, -1113.565]
  MoveL 553 to (43.78, 293.91, 260) mm, rotated rx 180 ry 0 rz -52.23 deg; joints [51.218, -26.302, 114.493, 51.232, 91.133, 91.41, -1117.765]
  MoveL 554 to (41.29, 296.51, 270) mm, rotated rx 180 ry 0 rz -48.51 deg; joints [50.872, -26.229, 114.011, 50.893, 91.399, 91.72, -1121.487]
  MoveL 555 to (39.03, 298.61, 280) mm, rotated rx -180 ry 0 rz -45.31 deg; joints [50.529, -26.148, 113.522, 50.558, 91.669, 92.028, -1124.686]
  MoveL 556 to (37.11, 300.24, 290) mm, rotated rx -180 ry 0 rz -42.69 deg; joints [50.189, -26.061, 113.024, 50.228, 91.944, 92.334, -1127.315]
  MoveL 557 to (43.85, 319.91, 290) mm, rotated rx 180 ry 0 rz -36.2 deg; joints [50.189, -24.747, 112.3, 50.214, 91.566, 91.88, -1133.803]
  Set speed (60.0 mm/s)
  MoveL 558 to (46.6, 317.98, 280) mm, rotated rx -180 ry 0 rz -38.79 deg; joints [50.529, -24.831, 112.796, 50.546, 91.293, 91.571, -1131.207]
  MoveL 559 to (49.86, 315.46, 270) mm, rotated rx -180 ry 0 rz -41.95 deg; joints [50.872, -24.908, 113.285, 50.883, 91.024, 91.259, -1128.046]
  MoveL 560 to (53.49, 312.31, 260) mm, rotated rx -180 ry 0 rz -45.64 deg; joints [51.218, -24.978, 113.766, 51.224, 90.759, 90.945, -1124.36]
  MoveL 561 to (57.36, 308.47, 250) mm, rotated rx -180 ry 0 rz -49.81 deg; joints [51.568, -25.042, 114.239, 51.571, 90.499, 90.629, -1120.194]
  MoveL 562 to (61.34, 303.9, 240) mm, rotated rx -180 ry 0 rz -54.41 deg; joints [51.921, -25.098, 114.704, 51.922, 90.243, 90.31, -1115.591]
  MoveL 563 to (65.27, 298.59, 230) mm, rotated rx -180 ry 0 rz -59.4 deg; joints [52.278, -25.148, 115.161, 52.278, 89.992, 89.989, -1110.596]
  MoveL 564 to (68.98, 292.54, 220) mm, rotated rx -180 ry 0 rz -64.75 deg; joints [52.638, -25.19, 115.61, 52.639, 89.745, 89.666, -1105.253]
  MoveL 565 to (72.31, 285.76, 210) mm, rotated rx -180 ry 0 rz -70.39 deg; joints [53.002, -25.225, 116.051, 53.005, 89.503, 89.34, -1099.605]
  MoveL 566 to (75.1, 278.3, 200) mm, rotated rx -180 ry 0 rz -76.3 deg; joints [53.369, -25.253, 116.485, 53.376, 89.265, 89.012, -1093.697]
  MoveL 567 to (77.2, 270.26, 190) mm, rotated rx -180 ry 0 rz -82.43 deg; joints [53.74, -25.275, 116.91, 53.751, 89.033, 88.682, -1087.571]
  MoveL 568 to (78.47, 261.74, 180) mm, rotated rx -180 ry 0 rz -88.73 deg; joints [54.114, -25.292, 117.329, 54.131, 88.806, 88.349, -1081.269]
  MoveL 569 to (78.79, 252.87, 170) mm, rotated rx -180 ry 0 rz -95.17 deg; joints [54.492, -25.304, 117.741, 54.517, 88.585, 88.016, -1074.829]
  MoveL 570 to (78.09, 243.82, 160) mm, rotated rx -180 ry 0 rz -101.71 deg; joints [54.874, -25.312, 118.147, 54.907, 88.37, 87.681, -1068.29]
  MoveL 571 to (76.31, 234.75, 150) mm, rotated rx 180 ry 0 rz -108.31 deg; joints [55.259, -25.318, 118.547, 55.301, 88.16, 87.346, -1061.689]
  MoveL 572 to (73.44, 225.85, 140) mm, rotated rx -180 ry 0 rz -114.94 deg; joints [55.647, -25.32, 118.941, 55.701, 87.958, 87.01, -1055.058]
  MoveL 573 to (69.5, 217.29, 130) mm, rotated rx -180 ry 0 rz -121.57 deg; joints [56.04, -25.322, 119.331, 56.105, 87.762, 86.674, -1048.432]
  MoveL 574 to (64.57, 209.26, 120) mm, rotated rx -180 ry 0 rz -128.16 deg; joints [56.436, -25.324, 119.716, 56.513, 87.573, 86.338, -1041.84]
  MoveL 575 to (58.74, 201.9, 110) mm, rotated rx -180 ry 0 rz -134.69 deg; joints [56.835, -25.326, 120.097, 56.926, 87.392, 86.003, -1035.313]
  MoveL 576 to (52.14, 195.34, 100) mm, rotated rx 180 ry 0 rz -141.12 deg; joints [57.239, -25.329, 120.475, 57.344, 87.218, 85.669, -1028.879]
  MoveL 577 to (44.91, 189.68, 90) mm, rotated rx -180 ry 0 rz -147.43 deg; joints [57.646, -25.333, 120.849, 57.766, 87.052, 85.337, -1022.567]
  MoveL 578 to (37.24, 184.98, 80) mm, rotated rx -180 ry 0 rz -153.6 deg; joints [58.056, -25.34, 121.22, 58.192, 86.893, 85.006, -1016.403]
  MoveL 579 to (29.3, 181.28, 70) mm, rotated rx -180 ry 0 rz -159.58 deg; joints [58.471, -25.348, 121.587, 58.622, 86.742, 84.676, -1010.416]
  MoveL 580 to (21.27, 178.55, 60) mm, rotated rx -180 ry 0 rz -165.37 deg; joints [58.889, -25.359, 121.952, 59.057, 86.599, 84.349, -1004.633]
  MoveL 581 to (13.31, 176.76, 50) mm, rotated rx -180 ry 0 rz -170.92 deg; joints [59.311, -25.372, 122.313, 59.496, 86.464, 84.024, -999.083]
  MoveL 582 to (5.58, 175.83, 40) mm, rotated rx -180 ry 0 rz -176.21 deg; joints [59.736, -25.386, 122.67, 59.938, 86.336, 83.7, -993.794]
  MoveL 583 to (-1.77, 175.65, 30) mm, rotated rx -180 ry 0 rz 178.8 deg; joints [60.166, -25.402, 123.024, 60.385, 86.217, 83.378, -988.796]
  MoveL 584 to (-8.64, 176.1, 20) mm, rotated rx -180 ry 0 rz 174.12 deg; joints [60.599, -25.418, 123.373, 60.835, 86.104, 83.059, -984.119]
  MoveL 585 to (-14.93, 177.06, 10) mm, rotated rx -180 ry 0 rz 169.79 deg; joints [61.035, -25.435, 123.718, 61.289, 85.999, 82.741, -979.795]
  MoveL 586 to (-20.57, 178.36, 0) mm, rotated rx -180 ry 0 rz 165.86 deg; joints [61.476, -25.451, 124.058, 61.747, 85.902, 82.424, -975.856]
  MoveL 587 to (43.85, 319.91, 290) mm, rotated rx -180 ry 0 rz -36.2 deg; joints [50.189, -24.747, 112.3, 50.214, 91.566, 91.88, -1133.803]
  Set speed (60.0 mm/s)
  MoveL 588 to (28.22, 306.19, 290) mm, rotated rx -180 ry 0 rz -31.42 deg; joints [50.189, -26.102, 113.046, 50.229, 91.956, 92.348, -1138.582]
  MoveL 589 to (-20.57, 178.36, 0) mm, rotated rx -180 ry 0 rz 165.86 deg; joints [61.476, -25.451, 124.058, 61.747, 85.902, 82.424, -975.856]
  Set speed (60.0 mm/s)
  MoveL 590 to (-10.16, 196.36, 0) mm, rotated rx -180 ry 0 rz 170.93 deg; joints [61.476, -26.912, 124.861, 61.707, 86.214, 83.006, -980.929]
  MoveL 591 to (-20.57, 178.36, 0) mm, rotated rx 180 ry 0 rz 165.86 deg; joints [61.476, -25.451, 124.058, 61.747, 85.902, 82.424, -975.856]
  Set speed (60.0 mm/s)
  MoveL 592 to (-14.93, 177.06, 10) mm, rotated rx -180 ry 0 rz 169.79 deg; joints [61.035, -25.435, 123.718, 61.289, 85.999, 82.741, -979.795]
  MoveL 593 to (-8.64, 176.1, 20) mm, rotated rx 180 ry 0 rz 174.12 deg; joints [60.599, -25.418, 123.373, 60.835, 86.104, 83.059, -984.119]
  MoveL 594 to (-1.77, 175.65, 30) mm, rotated rx -180 ry 0 rz 178.8 deg; joints [60.166, -25.402, 123.024, 60.385, 86.217, 83.378, -988.796]
  MoveL 595 to (5.58, 175.83, 40) mm, rotated rx -180 ry 0 rz -176.21 deg; joints [59.736, -25.386, 122.67, 59.938, 86.336, 83.7, -993.794]
  MoveL 596 to (13.31, 176.76, 50) mm, rotated rx -180 ry 0 rz -170.92 deg; joints [59.311, -25.372, 122.313, 59.496, 86.464, 84.024, -999.083]
  MoveL 597 to (21.27, 178.55, 60) mm, rotated rx -180 ry 0 rz -165.37 deg; joints [58.889, -25.359, 121.952, 59.057, 86.599, 84.349, -1004.633]
  MoveL 598 to (29.3, 181.28, 70) mm, rotated rx -180 ry 0 rz -159.58 deg; joints [58.471, -25.348, 121.587, 58.622, 86.742, 84.676, -1010.416]
  MoveL 599 to (37.24, 184.98, 80) mm, rotated rx -180 ry 0 rz -153.6 deg; joints [58.056, -25.34, 121.22, 58.192, 86.893, 85.006, -1016.403]
  MoveL 600 to (44.91, 189.68, 90) mm, rotated rx -180 ry 0 rz -147.43 deg; joints [57.646, -25.333, 120.849, 57.766, 87.052, 85.337, -1022.567]
  MoveL 601 to (52.14, 195.34, 100) mm, rotated rx -180 ry 0 rz -141.12 deg; joints [57.239, -25.329, 120.475, 57.344, 87.218, 85.669, -1028.879]
  MoveL 602 to (58.74, 201.9, 110) mm, rotated rx 180 ry 0 rz -134.69 deg; joints [56.835, -25.326, 120.097, 56.926, 87.392, 86.003, -1035.313]
  MoveL 603 to (64.57, 209.26, 120) mm, rotated rx -180 ry 0 rz -128.16 deg; joints [56.436, -25.324, 119.716, 56.513, 87.573, 86.338, -1041.84]
  MoveL 604 to (69.5, 217.29, 130) mm, rotated rx -180 ry 0 rz -121.57 deg; joints [56.04, -25.322, 119.331, 56.105, 87.762, 86.674, -1048.432]
  MoveL 605 to (73.44, 225.85, 140) mm, rotated rx -180 ry 0 rz -114.94 deg; joints [55.647, -25.32, 118.941, 55.701, 87.958, 87.01, -1055.058]
  MoveL 606 to (76.31, 234.75, 150) mm, rotated rx -180 ry 0 rz -108.31 deg; joints [55.259, -25.318, 118.547, 55.301, 88.16, 87.346, -1061.689]
  MoveL 607 to (78.09, 243.82, 160) mm, rotated rx -180 ry 0 rz -101.71 deg; joints [54.874, -25.312, 118.147, 54.907, 88.37, 87.681, -1068.29]
  MoveL 608 to (78.79, 252.87, 170) mm, rotated rx -180 ry 0 rz -95.17 deg; joints [54.492, -25.304, 117.741, 54.517, 88.585, 88.016, -1074.829]
  MoveL 609 to (78.47, 261.74, 180) mm, rotated rx -180 ry 0 rz -88.73 deg; joints [54.114, -25.292, 117.329, 54.131, 88.806, 88.349, -1081.269]
  MoveL 610 to (77.2, 270.26, 190) mm, rotated rx 180 ry 0 rz -82.43 deg; joints [53.74, -25.275, 116.91, 53.751, 89.033, 88.682, -1087.571]
  MoveL 611 to (75.1, 278.3, 200) mm, rotated rx -180 ry 0 rz -76.3 deg; joints [53.369, -25.253, 116.485, 53.376, 89.265, 89.012, -1093.697]
  MoveL 612 to (72.31, 285.76, 210) mm, rotated rx -180 ry 0 rz -70.39 deg; joints [53.002, -25.225, 116.051, 53.005, 89.503, 89.34, -1099.605]
  MoveL 613 to (68.98, 292.54, 220) mm, rotated rx 180 ry 0 rz -64.75 deg; joints [52.638, -25.19, 115.61, 52.639, 89.745, 89.666, -1105.253]
  MoveL 614 to (65.27, 298.59, 230) mm, rotated rx 180 ry 0 rz -59.4 deg; joints [52.278, -25.148, 115.161, 52.278, 89.992, 89.989, -1110.596]
  MoveL 615 to (61.34, 303.9, 240) mm, rotated rx -180 ry 0 rz -54.41 deg; joints [51.921, -25.098, 114.704, 51.922, 90.243, 90.31, -1115.591]
  MoveL 616 to (57.36, 308.47, 250) mm, rotated rx -180 ry 0 rz -49.81 deg; joints [51.568, -25.042, 114.239, 51.571, 90.499, 90.629, -1120.194]
  MoveL 617 to (53.49, 312.31, 260) mm, rotated rx -180 ry 0 rz -45.64 deg; joints [51.218, -24.978, 113.766, 51.224, 90.759, 90.945, -1124.36]
  MoveL 618 to (49.86, 315.46, 270) mm, rotated rx -180 ry 0 rz -41.95 deg; joints [50.872, -24.908, 113.285, 50.883, 91.024, 91.259, -1128.046]
  MoveL 619 to (46.6, 317.98, 280) mm, rotated rx -180 ry 0 rz -38.79 deg; joints [50.529, -24.831, 112.796, 50.546, 91.293, 91.571, -1131.207]
  MoveL 620 to (43.85, 319.91, 290) mm, rotated rx 180 ry 0 rz -36.2 deg; joints [50.189, -24.747, 112.3, 50.214, 91.566, 91.88, -1133.803]
  MoveL 621 to (28.22, 306.19, 290) mm, rotated rx -180 ry 0 rz -31.42 deg; joints [50.189, -26.102, 113.046, 50.229, 91.956, 92.348, -1138.582]
  Set speed (60.0 mm/s)
  MoveL 622 to (30.4, 304.94, 280) mm, rotated rx -180 ry 0 rz -34.08 deg; joints [50.529, -26.192, 113.545, 50.559, 91.682, 92.044, -1135.919]
  MoveL 623 to (33, 303.28, 270) mm, rotated rx -180 ry 0 rz -37.32 deg; joints [50.872, -26.275, 114.036, 50.893, 91.413, 91.737, -1132.679]
  MoveL 624 to (35.92, 301.18, 260) mm, rotated rx -180 ry 0 rz -41.09 deg; joints [51.218, -26.352, 114.52, 51.232, 91.147, 91.428, -1128.905]
  MoveL 625 to (39.07, 298.58, 250) mm, rotated rx -180 ry 0 rz -45.36 deg; joints [51.568, -26.422, 114.996, 51.577, 90.886, 91.117, -1124.643]
  MoveL 626 to (42.34, 295.45, 240) mm, rotated rx -180 ry 0 rz -50.06 deg; joints [51.921, -26.485, 115.464, 51.926, 90.63, 90.804, -1119.941]
  MoveL 627 to (45.62, 291.76, 230) mm, rotated rx -180 ry 0 rz -55.15 deg; joints [52.278, -26.54, 115.924, 52.28, 90.377, 90.487, -1114.846]
  MoveL 628 to (48.8, 287.5, 220) mm, rotated rx -180 ry 0 rz -60.59 deg; joints [52.638, -26.588, 116.376, 52.638, 90.129, 90.169, -1109.406]
  MoveL 629 to (51.74, 282.68, 210) mm, rotated rx 180 ry 0 rz -66.33 deg; joints [53.002, -26.629, 116.82, 53.002, 89.885, 89.848, -1103.668]
  MoveL 630 to (54.33, 277.32, 200) mm, rotated rx -180 ry 0 rz -72.32 deg; joints [53.369, -26.663, 117.257, 53.371, 89.646, 89.524, -1097.679]
  MoveL 631 to (56.44, 271.47, 190) mm, rotated rx -180 ry 0 rz -78.51 deg; joints [53.74, -26.691, 117.686, 53.744, 89.412, 89.198, -1091.486]
  MoveL 632 to (57.96, 265.2, 180) mm, rotated rx 180 ry 0 rz -84.87 deg; joints [54.114, -26.713, 118.107, 54.122, 89.183, 88.87, -1085.13]
  MoveL 633 to (58.8, 258.62, 170) mm, rotated rx -180 ry 0 rz -91.34 deg; joints [54.492, -26.73, 118.522, 54.505, 88.959, 88.541, -1078.655]
  MoveL 634 to (58.89, 251.83, 160) mm, rotated rx -180 ry 0 rz -97.9 deg; joints [54.874, -26.742, 118.931, 54.893, 88.741, 88.21, -1072.098]
  MoveL 635 to (58.18, 244.95, 150) mm, rotated rx 180 ry 0 rz -104.5 deg; joints [55.259, -26.751, 119.333, 55.286, 88.529, 87.878, -1065.497]
  MoveL 636 to (56.65, 238.12, 140) mm, rotated rx -180 ry 0 rz -111.11 deg; joints [55.647, -26.758, 119.73, 55.683, 88.323, 87.546, -1058.886]
  MoveL 637 to (54.3, 231.49, 130) mm, rotated rx 180 ry 0 rz -117.7 deg; joints [56.04, -26.763, 120.122, 56.085, 88.124, 87.213, -1052.295]
  MoveL 638 to (51.17, 225.17, 120) mm, rotated rx -180 ry 0 rz -124.24 deg; joints [56.436, -26.767, 120.509, 56.492, 87.932, 86.881, -1045.756]
  MoveL 639 to (47.33, 219.29, 110) mm, rotated rx -180 ry 0 rz -130.7 deg; joints [56.835, -26.772, 120.892, 56.903, 87.747, 86.549, -1039.296]
  MoveL 640 to (42.85, 213.95, 100) mm, rotated rx -180 ry 0 rz -137.06 deg; joints [57.239, -26.777, 121.271, 57.319, 87.57, 86.219, -1032.941]
  MoveL 641 to (37.86, 209.24, 90) mm, rotated rx 180 ry 0 rz -143.28 deg; joints [57.646, -26.783, 121.646, 57.739, 87.4, 85.889, -1026.718]
  MoveL 642 to (32.46, 205.23, 80) mm, rotated rx -180 ry 0 rz -149.35 deg; joints [58.056, -26.791, 122.018, 58.164, 87.237, 85.561, -1020.653]
  MoveL 643 to (26.8, 201.92, 70) mm, rotated rx -180 ry 0 rz -155.23 deg; joints [58.471, -26.801, 122.386, 58.592, 87.083, 85.235, -1014.769]
  MoveL 644 to (21, 199.35, 60) mm, rotated rx -180 ry 0 rz -160.91 deg; joints [58.889, -26.813, 122.751, 59.025, 86.936, 84.911, -1009.094]
  MoveL 645 to (15.19, 197.47, 50) mm, rotated rx -180 ry 0 rz -166.35 deg; joints [59.311, -26.827, 123.113, 59.462, 86.796, 84.588, -1003.653]
  MoveL 646 to (9.5, 196.25, 40) mm, rotated rx -180 ry 0 rz -171.53 deg; joints [59.736, -26.842, 123.471, 59.903, 86.665, 84.268, -998.473]
  MoveL 647 to (4.03, 195.62, 30) mm, rotated rx -180 ry 0 rz -176.42 deg; joints [60.166, -26.859, 123.825, 60.349, 86.541, 83.95, -993.581]
  MoveL 648 to (-1.12, 195.49, 20) mm, rotated rx -180 ry 0 rz 179.01 deg; joints [60.599, -26.877, 124.175, 60.798, 86.424, 83.633, -989.007]
  MoveL 649 to (-5.87, 195.78, 10) mm, rotated rx -180 ry 0 rz 174.78 deg; joints [61.035, -26.895, 124.521, 61.251, 86.315, 83.319, -984.779]
  MoveL 650 to (-10.16, 196.36, 0) mm, rotated rx -180 ry 0 rz 170.93 deg; joints [61.476, -26.912, 124.861, 61.707, 86.214, 83.006, -980.929]
  MoveL 651 to (28.22, 306.19, 290) mm, rotated rx -180 ry 0 rz -31.42 deg; joints [50.189, -26.102, 113.046, 50.229, 91.956, 92.348, -1138.582]
  Set speed (60.0 mm/s)
  MoveL 652 to (-21.11, 309.47, 290) mm, rotated rx -180 ry 0 rz 23.11 deg; joints [50.189, -26.125, 113.059, 50.229, 91.963, 92.356, -1193.11]
  MoveL 653 to (-10.16, 196.36, 0) mm, rotated rx 180 ry 0 rz 170.93 deg; joints [61.476, -26.912, 124.861, 61.707, 86.214, 83.006, -1340.929]
  Set speed (60.0 mm/s)
  MoveL 654 to (37.62, 209.05, 0) mm, rotated rx -180 ry 0 rz -143.56 deg; joints [61.476, -26.994, 124.905, 61.705, 86.232, 83.039, -1386.442]
  MoveL 655 to (-10.16, 196.36, 0) mm, rotated rx -180 ry 0 rz 170.93 deg; joints [61.476, -26.912, 124.861, 61.707, 86.214, 83.006, -1340.929]
  Set speed (60.0 mm/s)
  MoveL 656 to (-5.87, 195.78, 10) mm, rotated rx -180 ry 0 rz 174.78 deg; joints [61.035, -26.895, 124.521, 61.251, 86.315, 83.319, -1344.779]
  MoveL 657 to (-1.12, 195.49, 20) mm, rotated rx 180 ry 0 rz 179.01 deg; joints [60.599, -26.877, 124.175, 60.798, 86.424, 83.633, -1349.007]
  MoveL 658 to (4.03, 195.62, 30) mm, rotated rx -180 ry 0 rz -176.42 deg; joints [60.166, -26.859, 123.825, 60.349, 86.541, 83.95, -1353.581]
  MoveL 659 to (9.5, 196.25, 40) mm, rotated rx 180 ry 0 rz -171.53 deg; joints [59.736, -26.842, 123.471, 59.903, 86.665, 84.268, -1358.473]
  MoveL 660 to (15.19, 197.47, 50) mm, rotated rx -180 ry 0 rz -166.35 deg; joints [59.311, -26.827, 123.113, 59.462, 86.796, 84.588, -1363.653]
  MoveL 661 to (21, 199.35, 60) mm, rotated rx -180 ry 0 rz -160.91 deg; joints [58.889, -26.813, 122.751, 59.025, 86.936, 84.911, -1369.094]
  MoveL 662 to (26.8, 201.92, 70) mm, rotated rx -180 ry 0 rz -155.23 deg; joints [58.471, -26.801, 122.386, 58.592, 87.083, 85.235, -1374.769]
  MoveL 663 to (32.46, 205.23, 80) mm, rotated rx -180 ry 0 rz -149.35 deg; joints [58.056, -26.791, 122.018, 58.164, 87.237, 85.561, -1380.653]
  MoveL 664 to (37.86, 209.24, 90) mm, rotated rx -180 ry 0 rz -143.28 deg; joints [57.646, -26.783, 121.646, 57.739, 87.4, 85.889, -1386.718]
  MoveL 665 to (42.85, 213.95, 100) mm, rotated rx -180 ry 0 rz -137.06 deg; joints [57.239, -26.777, 121.271, 57.319, 87.57, 86.219, -1392.941]
  MoveL 666 to (47.33, 219.29, 110) mm, rotated rx -180 ry 0 rz -130.7 deg; joints [56.835, -26.772, 120.892, 56.903, 87.747, 86.549, -1399.296]
  MoveL 667 to (51.17, 225.17, 120) mm, rotated rx -180 ry 0 rz -124.24 deg; joints [56.436, -26.767, 120.509, 56.492, 87.932, 86.881, -1405.756]
  MoveL 668 to (54.3, 231.49, 130) mm, rotated rx -180 ry 0 rz -117.7 deg; joints [56.04, -26.763, 120.122, 56.085, 88.124, 87.213, -1412.295]
  MoveL 669 to (56.65, 238.12, 140) mm, rotated rx -180 ry 0 rz -111.11 deg; joints [55.647, -26.758, 119.73, 55.683, 88.323, 87.546, -1418.886]
  MoveL 670 to (58.18, 244.95, 150) mm, rotated rx 180 ry 0 rz -104.5 deg; joints [55.259, -26.751, 119.333, 55.286, 88.529, 87.878, -1425.497]
  MoveL 671 to (58.89, 251.83, 160) mm, rotated rx -180 ry 0 rz -97.9 deg; joints [54.874, -26.742, 118.931, 54.893, 88.741, 88.21, -1432.098]
  MoveL 672 to (58.8, 258.62, 170) mm, rotated rx -180 ry 0 rz -91.34 deg; joints [54.492, -26.73, 118.522, 54.505, 88.959, 88.541, -1438.655]
  MoveL 673 to (57.96, 265.2, 180) mm, rotated rx -180 ry 0 rz -84.87 deg; joints [54.114, -26.713, 118.107, 54.122, 89.183, 88.87, -1445.13]
